LIN {X 0,Y 312.586,Z 205.55,A -85,B 0,C 180,E1 -15727.528,E2 -15727.528} C_VEL
LIN {X 0,Y 312.637,Z 205.541,A -85,B 0,C 180,E1 -15731.656,E2 -15731.656} C_VEL
LIN {X 0,Y 312.692,Z 205.534,A -85,B 0,C 180,E1 -15735.685,E2 -15735.685} C_VEL
LIN {X 0,Y 312.7,Z 205.533,A -85,B 0,C 180,E1 -15739.641,E2 -15739.641} C_VEL
LIN {X 0,Y 312.87,Z 205.509,A -85,B 0,C 180,E1 -15742.253,E2 -15742.253} C_VEL
LIN {X 0,Y 312.716,Z 205.531,A -85,B 0,C 180,E1 -15744.842,E2 -15744.842} C_VEL
LIN {X 0,Y 312.988,Z 205.497,A -85,B 0,C 180,E1 -15748.712,E2 -15748.712} C_VEL
LIN {X 0,Y 312.988,Z 205.498,A -85,B 0,C 180,E1 -15751.286,E2 -15751.286} C_VEL
LIN {X 0,Y 312.713,Z 205.533,A -85,B 0,C 180,E1 -15755.157,E2 -15755.157} C_VEL
LIN {X 0,Y 312.862,Z 205.51,A -85,B 0,C 180,E1 -15757.745,E2 -15757.745} C_VEL
LIN {X 0,Y 312.665,Z 205.535,A -85,B 0,C 180,E1 -15761.67,E2 -15761.67} C_VEL
LIN {X 0,Y 312.696,Z 205.536,A -85,B 0,C 180,E1 -15764.887,E2 -15764.887} C_VEL
LIN {X 0,Y 312.626,Z 205.542,A -85,B 0,C 180,E1 -15769.236,E2 -15769.236} C_VEL
LIN {X 0,Y 312.541,Z 205.555,A -85,B 0,C 180,E1 -15772.789,E2 -15772.789} C_VEL
LIN {X 0,Y 312.577,Z 205.551,A -85,B 0,C 180,E1 -15776.722,E2 -15776.722} C_VEL
LIN {X 0,Y 312.539,Z 205.551,A -85,B 0,C 180,E1 -15779.649,E2 -15779.649} C_VEL
LIN {X 0,Y 312.513,Z 205.554,A -85,B 0,C 180,E1 -15783.688,E2 -15783.688} C_VEL
LIN {X 0,Y 312.546,Z 205.55,A -85,B 0,C 180,E1 -15787.381,E2 -15787.381} C_VEL
LIN {X 0,Y 312.526,Z 205.555,A -85,B 0,C 180,E1 -15790.702,E2 -15790.702} C_VEL
LIN {X 0,Y 312.528,Z 205.556,A -85,B 0,C 180,E1 -15794.194,E2 -15794.194} C_VEL
LIN {X 0,Y 312.526,Z 205.554,A -85,B 0,C 180,E1 -15797.908,E2 -15797.908} C_VEL
LIN {X 0,Y 312.549,Z 205.552,A -85,B 0,C 180,E1 -15801.905,E2 -15801.905} C_VEL
LIN {X 0,Y 312.499,Z 205.558,A -85,B 0,C 180,E1 -15805.79,E2 -15805.79} C_VEL
LIN {X 0,Y 312.493,Z 205.557,A -85,B 0,C 180,E1 -15806.992,E2 -15806.992} C_VEL
LIN {X 0,Y 311.844,Z 205.642,A -85,B 0,C 180,E1 -15808.068,E2 -15808.068} C_VEL
LIN {X 0,Y 309.031,Z 205.991,A -85,B 0,C 180,E1 -15809.82,E2 -15809.82} C_VEL
LIN {X 0,Y 306.634,Z 206.291,A -85,B 0,C 180,E1 -15811.24,E2 -15811.24} C_VEL
LIN {X 0,Y 305.599,Z 206.419,A -85,B 0,C 180,E1 -15812.339,E2 -15812.339} C_VEL
LIN {X 0,Y 305.511,Z 206.427,A -85,B 0,C 180,E1 -15812.712,E2 -15812.712} C_VEL
LIN {X 0,Y 305.5,Z 206.429,A -85,B 0,C 180,E1 -15815.539,E2 -15815.539} C_VEL
LIN {X 0,Y 305.511,Z 206.43,A -85,B 0,C 180,E1 -15819.815,E2 -15819.815} C_VEL
LIN {X 0,Y 305.567,Z 206.42,A -85,B 0,C 180,E1 -15822.603,E2 -15822.603} C_VEL
LIN {X 0,Y 305.641,Z 206.411,A -85,B 0,C 180,E1 -15825.349,E2 -15825.349} C_VEL
LIN {X 0,Y 305.628,Z 206.413,A -85,B 0,C 180,E1 -15829.4,E2 -15829.4} C_VEL
LIN {X 0,Y 305.789,Z 206.394,A -85,B 0,C 180,E1 -15832.074,E2 -15832.074} C_VEL
LIN {X 0,Y 305.679,Z 206.405,A -85,B 0,C 180,E1 -15834.724,E2 -15834.724} C_VEL
LIN {X 0,Y 305.949,Z 206.372,A -85,B 0,C 180,E1 -15838.684,E2 -15838.684} C_VEL
LIN {X 0,Y 305.949,Z 206.374,A -85,B 0,C 180,E1 -15841.317,E2 -15841.317} C_VEL
LIN {X 0,Y 305.844,Z 206.385,A -85,B 0,C 180,E1 -15846.598,E2 -15846.598} C_VEL
LIN {X 0,Y 305.729,Z 206.402,A -85,B 0,C 180,E1 -15849.261,E2 -15849.261} C_VEL
LIN {X 0,Y 305.582,Z 206.421,A -85,B 0,C 180,E1 -15853.297,E2 -15853.297} C_VEL
LIN {X 0,Y 305.588,Z 206.418,A -85,B 0,C 180,E1 -15856.021,E2 -15856.021} C_VEL
LIN {X 0,Y 305.571,Z 206.423,A -85,B 0,C 180,E1 -15859.446,E2 -15859.446} C_VEL
LIN {X 0,Y 305.485,Z 206.432,A -85,B 0,C 180,E1 -15863.043,E2 -15863.043} C_VEL
LIN {X 0,Y 305.52,Z 206.425,A -85,B 0,C 180,E1 -15866.22,E2 -15866.22} C_VEL
LIN {X 0,Y 305.483,Z 206.433,A -85,B 0,C 180,E1 -15869.049,E2 -15869.049} C_VEL
LIN {X 0,Y 305.437,Z 206.436,A -85,B 0,C 180,E1 -15871.954,E2 -15871.954} C_VEL
LIN {X 0,Y 305.458,Z 206.438,A -85,B 0,C 180,E1 -15875.114,E2 -15875.114} C_VEL
LIN {X 0,Y 305.436,Z 206.437,A -85,B 0,C 180,E1 -15878.528,E2 -15878.528} C_VEL
LIN {X 0,Y 305.451,Z 206.436,A -85,B 0,C 180,E1 -15882.587,E2 -15882.587} C_VEL
LIN {X 0,Y 305.422,Z 206.438,A -85,B 0,C 180,E1 -15886.346,E2 -15886.346} C_VEL
LIN {X 0,Y 305.456,Z 206.434,A -85,B 0,C 180,E1 -15889.894,E2 -15889.894} C_VEL
LIN {X 0,Y 305.478,Z 206.434,A -85,B 0,C 180,E1 -15893.633,E2 -15893.633} C_VEL
LIN {X 0,Y 305.536,Z 206.602,A -85,B 0,C 180,E1 -15895.711,E2 -15895.711} C_VEL
LIN {X 0,Y 309.119,Z 222.623,A -85,B 0,C 180,E1 -15899.555,E2 -15899.555} C_VEL
LIN {X 0,Y 311.405,Z 233.024,A -85,B 0,C 180,E1 -15901.938,E2 -15901.938} C_VEL
LIN {X 0,Y 310.895,Z 238.703,A -85,B 0,C 180,E1 -15903.122,E2 -15903.122} C_VEL
LIN {X 0,Y 308.443,Z 258.998,A -85,B 0,C 180,E1 -15907.254,E2 -15907.254} C_VEL
LIN {X 0,Y 310.83,Z 288.757,A -85,B 0,C 180,E1 -15908.249,E2 -15908.249} C_VEL
LIN {X 0,Y 311.426,Z 296.327,A -85,B 0,C 180,E1 -15908.49,E2 -15908.49} C_VEL
LIN {X 0,Y 309.963,Z 363.951,A -85,B 0,C 180,E1 -15910.377,E2 -15910.377} C_VEL
LIN {X 0,Y 309.194,Z 377.33,A -85,B 0,C 180,E1 -15911.016,E2 -15911.016} C_VEL
LIN {X 0,Y 308.473,Z 387.934,A -85,B 0,C 180,E1 -15911.745,E2 -15911.745} C_VEL
LIN {X 0,Y 307.527,Z 400.398,A -85,B 0,C 180,E1 -15912.889,E2 -15912.889} C_VEL
LIN {X 0,Y 306.587,Z 411.617,A -85,B 0,C 180,E1 -15914.219,E2 -15914.219} C_VEL
LIN {X 0,Y 305.71,Z 421.456,A -85,B 0,C 180,E1 -15915.693,E2 -15915.693} C_VEL
LIN {X 0,Y 304.983,Z 430.461,A -85,B 0,C 180,E1 -15917.356,E2 -15917.356} C_VEL
LIN {X 0,Y 304.502,Z 437.832,A -85,B 0,C 180,E1 -15919.024,E2 -15919.024} C_VEL
LIN {X 0,Y 304.218,Z 444.937,A -85,B 0,C 180,E1 -15921.03,E2 -15921.03} C_VEL
LIN {X 0,Y 304.201,Z 451.35,A -85,B 0,C 180,E1 -15923.368,E2 -15923.368} C_VEL
LIN {X 0,Y 304.234,Z 455.384,A -85,B 0,C 180,E1 -15925.363,E2 -15925.363} C_VEL
LIN {X 0,Y 304.425,Z 458.247,A -85,B 0,C 180,E1 -15927.355,E2 -15927.355} C_VEL
LIN {X 0,Y 304.502,Z 459.525,A -85,B 0,C 180,E1 -15928.678,E2 -15928.678} C_VEL
LIN {X 0,Y 304.466,Z 460.35,A -85,B 0,C 180,E1 -15930.001,E2 -15930.001} C_VEL
LIN {X 0,Y 304.461,Z 460.719,A -85,B 0,C 180,E1 -15931.324,E2 -15931.324} C_VEL
LIN {X 0,Y 304.248,Z 460.595,A -85,B 0,C 180,E1 -15932.649,E2 -15932.649} C_VEL
LIN {X 0,Y 304.007,Z 460.044,A -85,B 0,C 180,E1 -15933.978,E2 -15933.978} C_VEL
LIN {X 0,Y 303.954,Z 458.231,A -85,B 0,C 180,E1 -15936.146,E2 -15936.146} C_VEL
LIN {X 0,Y 304.006,Z 454.659,A -85,B 0,C 180,E1 -15938.643,E2 -15938.643} C_VEL
LIN {X 0,Y 304.327,Z 450.624,A -85,B 0,C 180,E1 -15940.647,E2 -15940.647} C_VEL
LIN {X 0,Y 305.295,Z 444.466,A -85,B 0,C 180,E1 -15942.971,E2 -15942.971} C_VEL
LIN {X 0,Y 306.481,Z 437.705,A -85,B 0,C 180,E1 -15944.951,E2 -15944.951} C_VEL
LIN {X 0,Y 307.994,Z 429.456,A -85,B 0,C 180,E1 -15946.881,E2 -15946.881} C_VEL
LIN {X 0,Y 309.674,Z 420.823,A -85,B 0,C 180,E1 -15948.526,E2 -15948.526} C_VEL
LIN {X 0,Y 311.798,Z 410.405,A -85,B 0,C 180,E1 -15950.106,E2 -15950.106} C_VEL
LIN {X 0,Y 313.859,Z 398.746,A -85,B 0,C 180,E1 -15951.511,E2 -15951.511} C_VEL
LIN {X 0,Y 315.687,Z 387.145,A -85,B 0,C 180,E1 -15952.584,E2 -15952.584} C_VEL
LIN {X 0,Y 317.519,Z 374.07,A -85,B 0,C 180,E1 -15953.48,E2 -15953.48} C_VEL
LIN {X 0,Y 318.763,Z 360.739,A -85,B 0,C 180,E1 -15954.116,E2 -15954.116} C_VEL
LIN {X 0,Y 320.717,Z 321.294,A -85,B 0,C 180,E1 -15955.308,E2 -15955.308} C_VEL
LIN {X 0,Y 321.751,Z 297.702,A -85,B 0,C 180,E1 -15956.035,E2 -15956.035} C_VEL
LIN {X 0,Y 320.348,Z 281.565,A -85,B 0,C 180,E1 -15956.817,E2 -15956.817} C_VEL
LIN {X 0,Y 317.918,Z 265.294,A -85,B 0,C 180,E1 -15957.783,E2 -15957.783} C_VEL
LIN {X 0,Y 316.106,Z 255.214,A -85,B 0,C 180,E1 -15958.474,E2 -15958.474} C_VEL
LIN {X 0,Y 317.384,Z 248.061,A -85,B 0,C 180,E1 -15959.917,E2 -15959.917} C_VEL
LIN {X 0,Y 317.312,Z 245.135,A -85,B 0,C 180,E1 -15960.626,E2 -15960.626} C_VEL
LIN {X 0,Y 315.192,Z 235.048,A -85,B 0,C 180,E1 -15963.495,E2 -15963.495} C_VEL
LIN {X 0,Y 313.001,Z 227.13,A -85,B 0,C 180,E1 -15966.066,E2 -15966.066} C_VEL
LIN {X 0,Y 310.682,Z 220.037,A -85,B 0,C 180,E1 -15968.7,E2 -15968.7} C_VEL
LIN {X 0,Y 307.74,Z 212.476,A -85,B 0,C 180,E1 -15972.079,E2 -15972.079} C_VEL
LIN {X 0,Y 306.8,Z 209.817,A -85,B 0,C 180,E1 -15973.411,E2 -15973.411} C_VEL
LIN {X 0,Y 305.434,Z 206.594,A -85,B 0,C 180,E1 -15975.345,E2 -15975.345} C_VEL
LIN {X 0,Y 305.444,Z 206.434,A -85,B 0,C 180,E1 -15978.143,E2 -15978.143} C_VEL
LIN {X 0,Y 305.471,Z 206.432,A -85,B 0,C 180,E1 -15981.596,E2 -15981.596} C_VEL
LIN {X 0,Y 305.466,Z 206.433,A -85,B 0,C 180,E1 -15984.887,E2 -15984.887} C_VEL
LIN {X 0,Y 305.453,Z 206.432,A -85,B 0,C 180,E1 -15988.356,E2 -15988.356} C_VEL
LIN {X 0,Y 305.516,Z 206.425,A -85,B 0,C 180,E1 -15991.113,E2 -15991.113} C_VEL
LIN {X 0,Y 305.574,Z 206.423,A -85,B 0,C 180,E1 -15994.088,E2 -15994.088} C_VEL
LIN {X 0,Y 305.503,Z 206.43,A -85,B 0,C 180,E1 -15998.402,E2 -15998.402} C_VEL
LIN {X 0,Y 305.628,Z 206.622,A -85,B 0,C 180,E1 -16001.48,E2 -16001.48} C_VEL
LIN {X 0,Y 307.294,Z 211.058,A -85,B 0,C 180,E1 -16004.07,E2 -16004.07} C_VEL
LIN {X 0,Y 309.466,Z 216.706,A -85,B 0,C 180,E1 -16006.873,E2 -16006.873} C_VEL
LIN {X 0,Y 312.183,Z 224.834,A -85,B 0,C 180,E1 -16010.279,E2 -16010.279} C_VEL
LIN {X 0,Y 313.959,Z 231.596,A -85,B 0,C 180,E1 -16012.728,E2 -16012.728} C_VEL
LIN {X 0,Y 315.055,Z 236.534,A -85,B 0,C 180,E1 -16014.298,E2 -16014.298} C_VEL
LIN {X 0,Y 318.008,Z 242.357,A -85,B 0,C 180,E1 -16015.047,E2 -16015.047} C_VEL
LIN {X 0,Y 321.331,Z 256.287,A -85,B 0,C 180,E1 -16016.159,E2 -16016.159} C_VEL
LIN {X 0,Y 322.892,Z 264.443,A -85,B 0,C 180,E1 -16016.718,E2 -16016.718} C_VEL
LIN {X 0,Y 319.31,Z 322.49,A -85,B 0,C 180,E1 -16018.738,E2 -16018.738} C_VEL
LIN {X 0,Y 318.441,Z 335.49,A -85,B 0,C 180,E1 -16019.446,E2 -16019.446} C_VEL
LIN {X 0,Y 317.313,Z 346.446,A -85,B 0,C 180,E1 -16020.278,E2 -16020.278} C_VEL
LIN {X 0,Y 315.87,Z 357.96,A -85,B 0,C 180,E1 -16021.434,E2 -16021.434} C_VEL
LIN {X 0,Y 314.377,Z 367.881,A -85,B 0,C 180,E1 -16022.722,E2 -16022.722} C_VEL
LIN {X 0,Y 312.691,Z 376.857,A -85,B 0,C 180,E1 -16024.188,E2 -16024.188} C_VEL
LIN {X 0,Y 311.231,Z 384.199,A -85,B 0,C 180,E1 -16025.696,E2 -16025.696} C_VEL
LIN {X 0,Y 309.642,Z 391.14,A -85,B 0,C 180,E1 -16027.498,E2 -16027.498} C_VEL
LIN {X 0,Y 308.405,Z 396.181,A -85,B 0,C 180,E1 -16029.178,E2 -16029.178} C_VEL
LIN {X 0,Y 307.203,Z 400.679,A -85,B 0,C 180,E1 -16031.146,E2 -16031.146} C_VEL
LIN {X 0,Y 306.147,Z 403.971,A -85,B 0,C 180,E1 -16033.271,E2 -16033.271} C_VEL
LIN {X 0,Y 305.491,Z 405.548,A -85,B 0,C 180,E1 -16034.93,E2 -16034.93} C_VEL
LIN {X 0,Y 305.155,Z 406.152,A -85,B 0,C 180,E1 -16036.043,E2 -16036.043} C_VEL
LIN {X 0,Y 304.79,Z 406.365,A -85,B 0,C 180,E1 -16037.442,E2 -16037.442} C_VEL
LIN {X 0,Y 304.567,Z 406,A -85,B 0,C 180,E1 -16038.898,E2 -16038.898} C_VEL
LIN {X 0,Y 304.389,Z 405.081,A -85,B 0,C 180,E1 -16040.262,E2 -16040.262} C_VEL
LIN {X 0,Y 304.389,Z 402.288,A -85,B 0,C 180,E1 -16042.548,E2 -16042.548} C_VEL
LIN {X 0,Y 304.598,Z 398.51,A -85,B 0,C 180,E1 -16044.538,E2 -16044.538} C_VEL
LIN {X 0,Y 304.972,Z 392.759,A -85,B 0,C 180,E1 -16046.703,E2 -16046.703} C_VEL
LIN {X 0,Y 305.379,Z 386.42,A -85,B 0,C 180,E1 -16048.524,E2 -16048.524} C_VEL
LIN {X 0,Y 305.989,Z 378.314,A -85,B 0,C 180,E1 -16050.35,E2 -16050.35} C_VEL
LIN {X 0,Y 306.664,Z 368.955,A -85,B 0,C 180,E1 -16052.01,E2 -16052.01} C_VEL
LIN {X 0,Y 307.327,Z 359.976,A -85,B 0,C 180,E1 -16053.286,E2 -16053.286} C_VEL
LIN {X 0,Y 308.049,Z 348.466,A -85,B 0,C 180,E1 -16054.576,E2 -16054.576} C_VEL
LIN {X 0,Y 308.666,Z 335.868,A -85,B 0,C 180,E1 -16055.633,E2 -16055.633} C_VEL
LIN {X 0,Y 309.157,Z 324.141,A -85,B 0,C 180,E1 -16056.332,E2 -16056.332} C_VEL
LIN {X 0,Y 309.352,Z 311.339,A -85,B 0,C 180,E1 -16056.837,E2 -16056.837} C_VEL
LIN {X 0,Y 310.809,Z 254.755,A -85,B 0,C 180,E1 -16058.574,E2 -16058.574} C_VEL
LIN {X 0,Y 307.658,Z 232.493,A -85,B 0,C 180,E1 -16059.453,E2 -16059.453} C_VEL
LIN {X 0,Y 308.195,Z 223.036,A -85,B 0,C 180,E1 -16061.836,E2 -16061.836} C_VEL
LIN {X 0,Y 307.872,Z 218.463,A -85,B 0,C 180,E1 -16063.072,E2 -16063.072} C_VEL
LIN {X 0,Y 305.51,Z 206.606,A -85,B 0,C 180,E1 -16066.507,E2 -16066.507} C_VEL
LIN {X 0,Y 305.457,Z 206.437,A -85,B 0,C 180,E1 -16069.892,E2 -16069.892} C_VEL
LIN {X 0,Y 305.48,Z 206.436,A -85,B 0,C 180,E1 -16073.631,E2 -16073.631} C_VEL
LIN {X 0,Y 305.464,Z 206.432,A -85,B 0,C 180,E1 -16076.482,E2 -16076.482} C_VEL
LIN {X 0,Y 305.463,Z 206.438,A -85,B 0,C 180,E1 -16079.59,E2 -16079.59} C_VEL
LIN {X 0,Y 305.52,Z 206.425,A -85,B 0,C 180,E1 -16082.608,E2 -16082.608} C_VEL
LIN {X 0,Y 305.507,Z 206.432,A -85,B 0,C 180,E1 -16085.538,E2 -16085.538} C_VEL
LIN {X 0,Y 305.518,Z 206.427,A -85,B 0,C 180,E1 -16089.814,E2 -16089.814} C_VEL
LIN {X 0,Y 305.573,Z 206.419,A -85,B 0,C 180,E1 -16092.602,E2 -16092.602} C_VEL
LIN {X 0,Y 305.647,Z 206.414,A -85,B 0,C 180,E1 -16095.348,E2 -16095.348} C_VEL
LIN {X 0,Y 305.637,Z 206.414,A -85,B 0,C 180,E1 -16099.399,E2 -16099.399} C_VEL
LIN {X 0,Y 305.811,Z 206.389,A -85,B 0,C 180,E1 -16102.073,E2 -16102.073} C_VEL
LIN {X 0,Y 305.688,Z 206.406,A -85,B 0,C 180,E1 -16104.723,E2 -16104.723} C_VEL
LIN {X 0,Y 305.955,Z 206.373,A -85,B 0,C 180,E1 -16108.683,E2 -16108.683} C_VEL
LIN {X 0,Y 305.955,Z 206.374,A -85,B 0,C 180,E1 -16111.315,E2 -16111.315} C_VEL
LIN {X 0,Y 305.684,Z 206.407,A -85,B 0,C 180,E1 -16115.276,E2 -16115.276} C_VEL
LIN {X 0,Y 305.804,Z 206.389,A -85,B 0,C 180,E1 -16117.925,E2 -16117.925} C_VEL
LIN {X 0,Y 305.6,Z 206.415,A -85,B 0,C 180,E1 -16121.944,E2 -16121.944} C_VEL
LIN {X 0,Y 305.633,Z 206.414,A -85,B 0,C 180,E1 -16125.034,E2 -16125.034} C_VEL
LIN {X 0,Y 305.572,Z 206.419,A -85,B 0,C 180,E1 -16129.444,E2 -16129.444} C_VEL
LIN {X 0,Y 305.485,Z 206.432,A -85,B 0,C 180,E1 -16133.041,E2 -16133.041} C_VEL
LIN {X 0,Y 305.548,Z 206.423,A -85,B 0,C 180,E1 -16136.229,E2 -16136.229} C_VEL
LIN {X 0,Y 305.49,Z 206.431,A -85,B 0,C 180,E1 -16139.049,E2 -16139.049} C_VEL
LIN {X 0,Y 305.438,Z 206.436,A -85,B 0,C 180,E1 -16141.951,E2 -16141.951} C_VEL
LIN {X 0,Y 305.457,Z 206.434,A -85,B 0,C 180,E1 -16145.112,E2 -16145.112} C_VEL
LIN {X 0,Y 305.487,Z 206.434,A -85,B 0,C 180,E1 -16148.539,E2 -16148.539} C_VEL
LIN {X 0,Y 305.502,Z 206.431,A -85,B 0,C 180,E1 -16152.596,E2 -16152.596} C_VEL
LIN {X 0,Y 305.48,Z 206.436,A -85,B 0,C 180,E1 -16156.356,E2 -16156.356} C_VEL
LIN {X 0,Y 305.459,Z 206.434,A -85,B 0,C 180,E1 -16159.893,E2 -16159.893} C_VEL
LIN {X 0,Y 305.495,Z 206.429,A -85,B 0,C 180,E1 -16163.626,E2 -16163.626} C_VEL
LIN {X 0,Y 305.428,Z 206.437,A -85,B 0,C 180,E1 -16166.983,E2 -16166.983} C_VEL
LIN {X 0,Y 305.513,Z 206.426,A -85,B 0,C 180,E1 -16171.114,E2 -16171.114} C_VEL
LIN {X 0,Y 305.511,Z 206.427,A -85,B 0,C 180,E1 -16172.712,E2 -16172.712} C_VEL
LIN {X 0,Y 304.826,Z 206.515,A -85,B 0,C 180,E1 -16173.813,E2 -16173.813} C_VEL
LIN {X 0,Y 301.945,Z 206.872,A -85,B 0,C 180,E1 -16175.604,E2 -16175.604} C_VEL
LIN {X 0,Y 299.516,Z 207.174,A -85,B 0,C 180,E1 -16177.058,E2 -16177.058} C_VEL
LIN {X 0,Y 298.486,Z 207.305,A -85,B 0,C 180,E1 -16178.184,E2 -16178.184} C_VEL
LIN {X 0,Y 298.408,Z 207.31,A -85,B 0,C 180,E1 -16178.566,E2 -16178.566} C_VEL
LIN {X 0,Y 298.53,Z 207.299,A -85,B 0,C 180,E1 -16182.18,E2 -16182.18} C_VEL
LIN {X 0,Y 298.585,Z 207.288,A -85,B 0,C 180,E1 -16184.995,E2 -16184.995} C_VEL
LIN {X 0,Y 298.584,Z 207.29,A -85,B 0,C 180,E1 -16189.147,E2 -16189.147} C_VEL
LIN {X 0,Y 298.734,Z 207.275,A -85,B 0,C 180,E1 -16191.886,E2 -16191.886} C_VEL
LIN {X 0,Y 298.649,Z 207.281,A -85,B 0,C 180,E1 -16194.599,E2 -16194.599} C_VEL
LIN {X 0,Y 298.916,Z 207.248,A -85,B 0,C 180,E1 -16198.653,E2 -16198.653} C_VEL
LIN {X 0,Y 298.916,Z 207.25,A -85,B 0,C 180,E1 -16201.348,E2 -16201.348} C_VEL
LIN {X 0,Y 298.79,Z 207.264,A -85,B 0,C 180,E1 -16206.755,E2 -16206.755} C_VEL
LIN {X 0,Y 298.674,Z 207.283,A -85,B 0,C 180,E1 -16209.481,E2 -16209.481} C_VEL
LIN {X 0,Y 298.546,Z 207.298,A -85,B 0,C 180,E1 -16213.616,E2 -16213.616} C_VEL
LIN {X 0,Y 298.543,Z 207.294,A -85,B 0,C 180,E1 -16216.41,E2 -16216.41} C_VEL
LIN {X 0,Y 298.506,Z 207.301,A -85,B 0,C 180,E1 -16219.656,E2 -16219.656} C_VEL
LIN {X 0,Y 298.452,Z 207.308,A -85,B 0,C 180,E1 -16223.599,E2 -16223.599} C_VEL
LIN {X 0,Y 298.48,Z 207.302,A -85,B 0,C 180,E1 -16226.576,E2 -16226.576} C_VEL
LIN {X 0,Y 298.412,Z 207.313,A -85,B 0,C 180,E1 -16229.643,E2 -16229.643} C_VEL
LIN {X 0,Y 298.39,Z 207.315,A -85,B 0,C 180,E1 -16232.802,E2 -16232.802} C_VEL
LIN {X 0,Y 298.44,Z 207.31,A -85,B 0,C 180,E1 -16236.808,E2 -16236.808} C_VEL
LIN {X 0,Y 298.384,Z 207.319,A -85,B 0,C 180,E1 -16241.089,E2 -16241.089} C_VEL
LIN {X 0,Y 298.396,Z 207.317,A -85,B 0,C 180,E1 -16243.105,E2 -16243.105} C_VEL
LIN {X 0,Y 298.4,Z 207.317,A -85,B 0,C 180,E1 -16246.922,E2 -16246.922} C_VEL
LIN {X 0,Y 298.397,Z 207.317,A -85,B 0,C 180,E1 -16251.009,E2 -16251.009} C_VEL
LIN {X 0,Y 298.436,Z 207.312,A -85,B 0,C 180,E1 -16254.765,E2 -16254.765} C_VEL
LIN {X 0,Y 298.504,Z 207.599,A -85,B 0,C 180,E1 -16255.383,E2 -16255.383} C_VEL
LIN {X 0,Y 302.006,Z 223.143,A -85,B 0,C 180,E1 -16259.207,E2 -16259.207} C_VEL
LIN {X 0,Y 304.454,Z 234.529,A -85,B 0,C 180,E1 -16261.874,E2 -16261.874} C_VEL
LIN {X 0,Y 302.813,Z 247.876,A -85,B 0,C 180,E1 -16264.691,E2 -16264.691} C_VEL
LIN {X 0,Y 301.499,Z 258.879,A -85,B 0,C 180,E1 -16266.956,E2 -16266.956} C_VEL
LIN {X 0,Y 304.053,Z 291.047,A -85,B 0,C 180,E1 -16268.044,E2 -16268.044} C_VEL
LIN {X 0,Y 304.463,Z 297.206,A -85,B 0,C 180,E1 -16268.245,E2 -16268.245} C_VEL
LIN {X 0,Y 303.009,Z 362.838,A -85,B 0,C 180,E1 -16270.128,E2 -16270.128} C_VEL
LIN {X 0,Y 302.298,Z 375.668,A -85,B 0,C 180,E1 -16270.742,E2 -16270.742} C_VEL
LIN {X 0,Y 301.46,Z 387.599,A -85,B 0,C 180,E1 -16271.569,E2 -16271.569} C_VEL
LIN {X 0,Y 300.569,Z 399.224,A -85,B 0,C 180,E1 -16272.656,E2 -16272.656} C_VEL
LIN {X 0,Y 299.668,Z 409.89,A -85,B 0,C 180,E1 -16273.927,E2 -16273.927} C_VEL
LIN {X 0,Y 298.749,Z 419.496,A -85,B 0,C 180,E1 -16275.352,E2 -16275.352} C_VEL
LIN {X 0,Y 298.014,Z 428.729,A -85,B 0,C 180,E1 -16277.055,E2 -16277.055} C_VEL
LIN {X 0,Y 297.505,Z 436.289,A -85,B 0,C 180,E1 -16278.763,E2 -16278.763} C_VEL
LIN {X 0,Y 297.167,Z 443.62,A -85,B 0,C 180,E1 -16280.815,E2 -16280.815} C_VEL
LIN {X 0,Y 297.111,Z 448.509,A -85,B 0,C 180,E1 -16282.526,E2 -16282.526} C_VEL
LIN {X 0,Y 297.158,Z 453.096,A -85,B 0,C 180,E1 -16284.573,E2 -16284.573} C_VEL
LIN {X 0,Y 297.233,Z 455.45,A -85,B 0,C 180,E1 -16285.933,E2 -16285.933} C_VEL
LIN {X 0,Y 297.357,Z 457.329,A -85,B 0,C 180,E1 -16287.292,E2 -16287.292} C_VEL
LIN {X 0,Y 297.458,Z 458.678,A -85,B 0,C 180,E1 -16288.647,E2 -16288.647} C_VEL
LIN {X 0,Y 297.424,Z 459.55,A -85,B 0,C 180,E1 -16290.001,E2 -16290.001} C_VEL
LIN {X 0,Y 297.412,Z 459.991,A -85,B 0,C 180,E1 -16291.355,E2 -16291.355} C_VEL
LIN {X 0,Y 297.18,Z 459.924,A -85,B 0,C 180,E1 -16292.712,E2 -16292.712} C_VEL
LIN {X 0,Y 296.892,Z 458.511,A -85,B 0,C 180,E1 -16295.434,E2 -16295.434} C_VEL
LIN {X 0,Y 296.856,Z 457.15,A -85,B 0,C 180,E1 -16296.799,E2 -16296.799} C_VEL
LIN {X 0,Y 296.944,Z 454.273,A -85,B 0,C 180,E1 -16298.85,E2 -16298.85} C_VEL
LIN {X 0,Y 297.288,Z 450.333,A -85,B 0,C 180,E1 -16300.902,E2 -16300.902} C_VEL
LIN {X 0,Y 298.193,Z 445.244,A -85,B 0,C 180,E1 -16302.939,E2 -16302.939} C_VEL
LIN {X 0,Y 299.623,Z 437.706,A -85,B 0,C 180,E1 -16305.301,E2 -16305.301} C_VEL
LIN {X 0,Y 301.233,Z 429.528,A -85,B 0,C 180,E1 -16307.306,E2 -16307.306} C_VEL
LIN {X 0,Y 302.974,Z 421.216,A -85,B 0,C 180,E1 -16308.951,E2 -16308.951} C_VEL
LIN {X 0,Y 305.182,Z 411.1,A -85,B 0,C 180,E1 -16310.561,E2 -16310.561} C_VEL
LIN {X 0,Y 307.33,Z 399.712,A -85,B 0,C 180,E1 -16311.992,E2 -16311.992} C_VEL
LIN {X 0,Y 309.22,Z 388.71,A -85,B 0,C 180,E1 -16313.084,E2 -16313.084} C_VEL
LIN {X 0,Y 310.935,Z 377.678,A -85,B 0,C 180,E1 -16313.919,E2 -16313.919} C_VEL
LIN {X 0,Y 312.486,Z 364.01,A -85,B 0,C 180,E1 -16314.676,E2 -16314.676} C_VEL
LIN {X 0,Y 313.348,Z 350.32,A -85,B 0,C 180,E1 -16315.18,E2 -16315.18} C_VEL
LIN {X 0,Y 316.005,Z 299.425,A -85,B 0,C 180,E1 -16316.714,E2 -16316.714} C_VEL
LIN {X 0,Y 314.757,Z 283.698,A -85,B 0,C 180,E1 -16317.507,E2 -16317.507} C_VEL
LIN {X 0,Y 312.523,Z 267.935,A -85,B 0,C 180,E1 -16318.473,E2 -16318.473} C_VEL
LIN {X 0,Y 310.227,Z 254.673,A -85,B 0,C 180,E1 -16319.427,E2 -16319.427} C_VEL
LIN {X 0,Y 311.077,Z 249.985,A -85,B 0,C 180,E1 -16320.401,E2 -16320.401} C_VEL
LIN {X 0,Y 310.754,Z 246.429,A -85,B 0,C 180,E1 -16321.344,E2 -16321.344} C_VEL
LIN {X 0,Y 308.655,Z 236.658,A -85,B 0,C 180,E1 -16324.283,E2 -16324.283} C_VEL
LIN {X 0,Y 306.72,Z 229.655,A -85,B 0,C 180,E1 -16326.681,E2 -16326.681} C_VEL
LIN {X 0,Y 304.675,Z 223.49,A -85,B 0,C 180,E1 -16329.095,E2 -16329.095} C_VEL
LIN {X 0,Y 301.952,Z 216.305,A -85,B 0,C 180,E1 -16332.453,E2 -16332.453} C_VEL
LIN {X 0,Y 301.133,Z 213.981,A -85,B 0,C 180,E1 -16333.655,E2 -16333.655} C_VEL
LIN {X 0,Y 299.322,Z 210.079,A -85,B 0,C 180,E1 -16336.16,E2 -16336.16} C_VEL
LIN {X 0,Y 298.402,Z 207.38,A -85,B 0,C 180,E1 -16338.29,E2 -16338.29} C_VEL
LIN {X 0,Y 298.412,Z 207.31,A -85,B 0,C 180,E1 -16342.241,E2 -16342.241} C_VEL
LIN {X 0,Y 298.412,Z 207.313,A -85,B 0,C 180,E1 -16345.581,E2 -16345.581} C_VEL
LIN {X 0,Y 298.395,Z 207.311,A -85,B 0,C 180,E1 -16348.79,E2 -16348.79} C_VEL
LIN {X 0,Y 298.462,Z 207.309,A -85,B 0,C 180,E1 -16351.904,E2 -16351.904} C_VEL
LIN {X 0,Y 298.489,Z 207.3,A -85,B 0,C 180,E1 -16354.924,E2 -16354.924} C_VEL
LIN {X 0,Y 298.493,Z 207.498,A -85,B 0,C 180,E1 -16358.686,E2 -16358.686} C_VEL
LIN {X 0,Y 300.11,Z 211.303,A -85,B 0,C 180,E1 -16361.569,E2 -16361.569} C_VEL
LIN {X 0,Y 302.043,Z 216.312,A -85,B 0,C 180,E1 -16364.523,E2 -16364.523} C_VEL
LIN {X 0,Y 304.188,Z 222.326,A -85,B 0,C 180,E1 -16367.482,E2 -16367.482} C_VEL
LIN {X 0,Y 306.717,Z 230.133,A -85,B 0,C 180,E1 -16370.77,E2 -16370.77} C_VEL
LIN {X 0,Y 308.263,Z 236.949,A -85,B 0,C 180,E1 -16373.166,E2 -16373.166} C_VEL
LIN {X 0,Y 312.996,Z 246.172,A -85,B 0,C 180,E1 -16374.447,E2 -16374.447} C_VEL
LIN {X 0,Y 316.43,Z 261.566,A -85,B 0,C 180,E1 -16375.681,E2 -16375.681} C_VEL
LIN {X 0,Y 317.142,Z 266.341,A -85,B 0,C 180,E1 -16376.003,E2 -16376.003} C_VEL
LIN {X 0,Y 313.423,Z 323.086,A -85,B 0,C 180,E1 -16378.032,E2 -16378.032} C_VEL
LIN {X 0,Y 312.507,Z 335.54,A -85,B 0,C 180,E1 -16378.711,E2 -16378.711} C_VEL
LIN {X 0,Y 311.419,Z 346.158,A -85,B 0,C 180,E1 -16379.514,E2 -16379.514} C_VEL
LIN {X 0,Y 309.914,Z 357.516,A -85,B 0,C 180,E1 -16380.651,E2 -16380.651} C_VEL
LIN {X 0,Y 308.272,Z 367.589,A -85,B 0,C 180,E1 -16381.959,E2 -16381.959} C_VEL
LIN {X 0,Y 306.67,Z 375.822,A -85,B 0,C 180,E1 -16383.284,E2 -16383.284} C_VEL
LIN {X 0,Y 304.928,Z 384.109,A -85,B 0,C 180,E1 -16384.958,E2 -16384.958} C_VEL
LIN {X 0,Y 303.405,Z 390.75,A -85,B 0,C 180,E1 -16386.65,E2 -16386.65} C_VEL
LIN {X 0,Y 301.718,Z 396.95,A -85,B 0,C 180,E1 -16388.708,E2 -16388.708} C_VEL
LIN {X 0,Y 300.367,Z 401.538,A -85,B 0,C 180,E1 -16390.788,E2 -16390.788} C_VEL
LIN {X 0,Y 299.629,Z 403.785,A -85,B 0,C 180,E1 -16392.186,E2 -16392.186} C_VEL
LIN {X 0,Y 298.956,Z 405.444,A -85,B 0,C 180,E1 -16393.596,E2 -16393.596} C_VEL
LIN {X 0,Y 298.411,Z 406.575,A -85,B 0,C 180,E1 -16395.069,E2 -16395.069} C_VEL
LIN {X 0,Y 297.972,Z 407.048,A -85,B 0,C 180,E1 -16396.441,E2 -16396.441} C_VEL
LIN {X 0,Y 297.645,Z 406.99,A -85,B 0,C 180,E1 -16397.875,E2 -16397.875} C_VEL
LIN {X 0,Y 297.423,Z 406.355,A -85,B 0,C 180,E1 -16399.318,E2 -16399.318} C_VEL
LIN {X 0,Y 297.288,Z 405.106,A -85,B 0,C 180,E1 -16400.769,E2 -16400.769} C_VEL
LIN {X 0,Y 297.317,Z 402.372,A -85,B 0,C 180,E1 -16402.796,E2 -16402.796} C_VEL
LIN {X 0,Y 297.495,Z 399.257,A -85,B 0,C 180,E1 -16404.419,E2 -16404.419} C_VEL
LIN {X 0,Y 297.872,Z 393.545,A -85,B 0,C 180,E1 -16406.633,E2 -16406.633} C_VEL
LIN {X 0,Y 298.292,Z 387.243,A -85,B 0,C 180,E1 -16408.496,E2 -16408.496} C_VEL
LIN {X 0,Y 298.889,Z 379.151,A -85,B 0,C 180,E1 -16410.367,E2 -16410.367} C_VEL
LIN {X 0,Y 299.488,Z 371.033,A -85,B 0,C 180,E1 -16411.87,E2 -16411.87} C_VEL
LIN {X 0,Y 300.259,Z 360.929,A -85,B 0,C 180,E1 -16413.37,E2 -16413.37} C_VEL
LIN {X 0,Y 300.983,Z 349.663,A -85,B 0,C 180,E1 -16414.673,E2 -16414.673} C_VEL
LIN {X 0,Y 301.568,Z 338.856,A -85,B 0,C 180,E1 -16415.634,E2 -16415.634} C_VEL
LIN {X 0,Y 302.117,Z 326.182,A -85,B 0,C 180,E1 -16416.461,E2 -16416.461} C_VEL
LIN {X 0,Y 302.408,Z 313.068,A -85,B 0,C 180,E1 -16417.017,E2 -16417.017} C_VEL
LIN {X 0,Y 303.881,Z 255.418,A -85,B 0,C 180,E1 -16418.843,E2 -16418.843} C_VEL
LIN {X 0,Y 300.689,Z 232.571,A -85,B 0,C 180,E1 -16419.784,E2 -16419.784} C_VEL
LIN {X 0,Y 301.231,Z 221.891,A -85,B 0,C 180,E1 -16422.577,E2 -16422.577} C_VEL
LIN {X 0,Y 298.913,Z 209.734,A -85,B 0,C 180,E1 -16426.084,E2 -16426.084} C_VEL
LIN {X 0,Y 298.496,Z 207.637,A -85,B 0,C 180,E1 -16426.729,E2 -16426.729} C_VEL
LIN {X 0,Y 298.467,Z 207.336,A -85,B 0,C 180,E1 -16426.932,E2 -16426.932} C_VEL
LIN {X 0,Y 298.403,Z 207.313,A -85,B 0,C 180,E1 -16431.005,E2 -16431.005} C_VEL
LIN {X 0,Y 298.417,Z 207.313,A -85,B 0,C 180,E1 -16433.929,E2 -16433.929} C_VEL
LIN {X 0,Y 298.395,Z 207.315,A -85,B 0,C 180,E1 -16437.982,E2 -16437.982} C_VEL
LIN {X 0,Y 298.462,Z 207.307,A -85,B 0,C 180,E1 -16441.903,E2 -16441.903} C_VEL
LIN {X 0,Y 298.484,Z 207.303,A -85,B 0,C 180,E1 -16444.923,E2 -16444.923} C_VEL
LIN {X 0,Y 298.449,Z 207.311,A -85,B 0,C 180,E1 -16449.314,E2 -16449.314} C_VEL
LIN {X 0,Y 298.536,Z 207.295,A -85,B 0,C 180,E1 -16452.178,E2 -16452.178} C_VEL
LIN {X 0,Y 298.592,Z 207.29,A -85,B 0,C 180,E1 -16454.994,E2 -16454.994} C_VEL
LIN {X 0,Y 298.592,Z 207.293,A -85,B 0,C 180,E1 -16459.146,E2 -16459.146} C_VEL
LIN {X 0,Y 298.756,Z 207.268,A -85,B 0,C 180,E1 -16461.885,E2 -16461.885} C_VEL
LIN {X 0,Y 298.658,Z 207.281,A -85,B 0,C 180,E1 -16464.598,E2 -16464.598} C_VEL
LIN {X 0,Y 298.921,Z 207.249,A -85,B 0,C 180,E1 -16468.652,E2 -16468.652} C_VEL
LIN {X 0,Y 298.921,Z 207.25,A -85,B 0,C 180,E1 -16471.346,E2 -16471.346} C_VEL
LIN {X 0,Y 298.788,Z 207.267,A -85,B 0,C 180,E1 -16476.753,E2 -16476.753} C_VEL
LIN {X 0,Y 298.677,Z 207.279,A -85,B 0,C 180,E1 -16479.48,E2 -16479.48} C_VEL
LIN {X 0,Y 298.548,Z 207.294,A -85,B 0,C 180,E1 -16483.614,E2 -16483.614} C_VEL
LIN {X 0,Y 298.544,Z 207.295,A -85,B 0,C 180,E1 -16486.408,E2 -16486.408} C_VEL
LIN {X 0,Y 298.507,Z 207.299,A -85,B 0,C 180,E1 -16489.654,E2 -16489.654} C_VEL
LIN {X 0,Y 298.452,Z 207.305,A -85,B 0,C 180,E1 -16493.597,E2 -16493.597} C_VEL
LIN {X 0,Y 298.486,Z 207.305,A -85,B 0,C 180,E1 -16496.573,E2 -16496.573} C_VEL
LIN {X 0,Y 298.415,Z 207.31,A -85,B 0,C 180,E1 -16499.64,E2 -16499.64} C_VEL
LIN {X 0,Y 298.389,Z 207.316,A -85,B 0,C 180,E1 -16502.799,E2 -16502.799} C_VEL
LIN {X 0,Y 298.464,Z 207.307,A -85,B 0,C 180,E1 -16506.813,E2 -16506.813} C_VEL
LIN {X 0,Y 298.448,Z 207.306,A -85,B 0,C 180,E1 -16511.102,E2 -16511.102} C_VEL
LIN {X 0,Y 298.452,Z 207.306,A -85,B 0,C 180,E1 -16513.115,E2 -16513.115} C_VEL
LIN {X 0,Y 298.428,Z 207.309,A -85,B 0,C 180,E1 -16516.926,E2 -16516.926} C_VEL
LIN {X 0,Y 298.424,Z 207.309,A -85,B 0,C 180,E1 -16520.999,E2 -16520.999} C_VEL
LIN {X 0,Y 298.427,Z 207.311,A -85,B 0,C 180,E1 -16523.932,E2 -16523.932} C_VEL
LIN {X 0,Y 298.392,Z 207.316,A -85,B 0,C 180,E1 -16527.982,E2 -16527.982} C_VEL
LIN {X 0,Y 298.456,Z 207.308,A -85,B 0,C 180,E1 -16531.904,E2 -16531.904} C_VEL
LIN {X 0,Y 298.478,Z 207.302,A -85,B 0,C 180,E1 -16534.924,E2 -16534.924} C_VEL
LIN {X 0,Y 298.408,Z 207.31,A -85,B 0,C 180,E1 -16538.566,E2 -16538.566} C_VEL
LIN {X 0,Y 297.753,Z 207.396,A -85,B 0,C 180,E1 -16539.692,E2 -16539.692} C_VEL
LIN {X 0,Y 294.911,Z 207.749,A -85,B 0,C 180,E1 -16541.528,E2 -16541.528} C_VEL
LIN {X 0,Y 292.538,Z 208.042,A -85,B 0,C 180,E1 -16543.018,E2 -16543.018} C_VEL
LIN {X 0,Y 291.584,Z 208.163,A -85,B 0,C 180,E1 -16544.171,E2 -16544.171} C_VEL
LIN {X 0,Y 291.541,Z 208.166,A -85,B 0,C 180,E1 -16544.561,E2 -16544.561} C_VEL
LIN {X 0,Y 291.528,Z 208.168,A -85,B 0,C 180,E1 -16548.881,E2 -16548.881} C_VEL
LIN {X 0,Y 291.681,Z 208.153,A -85,B 0,C 180,E1 -16551.688,E2 -16551.688} C_VEL
LIN {X 0,Y 291.62,Z 208.157,A -85,B 0,C 180,E1 -16554.469,E2 -16554.469} C_VEL
LIN {X 0,Y 291.882,Z 208.124,A -85,B 0,C 180,E1 -16558.621,E2 -16558.621} C_VEL
LIN {X 0,Y 291.882,Z 208.126,A -85,B 0,C 180,E1 -16561.38,E2 -16561.38} C_VEL
LIN {X 0,Y 291.739,Z 208.143,A -85,B 0,C 180,E1 -16566.919,E2 -16566.919} C_VEL
LIN {X 0,Y 291.623,Z 208.159,A -85,B 0,C 180,E1 -16569.713,E2 -16569.713} C_VEL
LIN {X 0,Y 291.516,Z 208.171,A -85,B 0,C 180,E1 -16573.951,E2 -16573.951} C_VEL
LIN {X 0,Y 291.481,Z 208.175,A -85,B 0,C 180,E1 -16576.819,E2 -16576.819} C_VEL
LIN {X 0,Y 291.445,Z 208.179,A -85,B 0,C 180,E1 -16579.876,E2 -16579.876} C_VEL
LIN {X 0,Y 291.394,Z 208.185,A -85,B 0,C 180,E1 -16584.206,E2 -16584.206} C_VEL
LIN {X 0,Y 291.414,Z 208.187,A -85,B 0,C 180,E1 -16587.273,E2 -16587.273} C_VEL
LIN {X 0,Y 291.33,Z 208.193,A -85,B 0,C 180,E1 -16590.438,E2 -16590.438} C_VEL
LIN {X 0,Y 291.34,Z 208.193,A -85,B 0,C 180,E1 -16593.7,E2 -16593.7} C_VEL
LIN {X 0,Y 291.368,Z 208.192,A -85,B 0,C 180,E1 -16597.254,E2 -16597.254} C_VEL
LIN {X 0,Y 291.329,Z 208.195,A -85,B 0,C 180,E1 -16600.644,E2 -16600.644} C_VEL
LIN {X 0,Y 291.287,Z 208.199,A -85,B 0,C 180,E1 -16604.403,E2 -16604.403} C_VEL
LIN {X 0,Y 291.324,Z 208.195,A -85,B 0,C 180,E1 -16608.406,E2 -16608.406} C_VEL
LIN {X 0,Y 291.346,Z 208.195,A -85,B 0,C 180,E1 -16611.159,E2 -16611.159} C_VEL
LIN {X 0,Y 291.417,Z 208.319,A -85,B 0,C 180,E1 -16614.957,E2 -16614.957} C_VEL
LIN {X 0,Y 294.6,Z 222.569,A -85,B 0,C 180,E1 -16618.583,E2 -16618.583} C_VEL
LIN {X 0,Y 297.158,Z 234.002,A -85,B 0,C 180,E1 -16621.345,E2 -16621.345} C_VEL
LIN {X 0,Y 297.474,Z 235.968,A -85,B 0,C 180,E1 -16621.804,E2 -16621.804} C_VEL
LIN {X 0,Y 294.864,Z 255.874,A -85,B 0,C 180,E1 -16626.098,E2 -16626.098} C_VEL
LIN {X 0,Y 294.548,Z 258.705,A -85,B 0,C 180,E1 -16626.635,E2 -16626.635} C_VEL
LIN {X 0,Y 297.025,Z 290.847,A -85,B 0,C 180,E1 -16627.756,E2 -16627.756} C_VEL
LIN {X 0,Y 297.514,Z 297.833,A -85,B 0,C 180,E1 -16627.99,E2 -16627.99} C_VEL
LIN {X 0,Y 296.009,Z 362.76,A -85,B 0,C 180,E1 -16629.909,E2 -16629.909} C_VEL
LIN {X 0,Y 295.297,Z 375.434,A -85,B 0,C 180,E1 -16630.538,E2 -16630.538} C_VEL
LIN {X 0,Y 294.436,Z 387.253,A -85,B 0,C 180,E1 -16631.383,E2 -16631.383} C_VEL
LIN {X 0,Y 293.47,Z 399.621,A -85,B 0,C 180,E1 -16632.583,E2 -16632.583} C_VEL
LIN {X 0,Y 292.502,Z 410.674,A -85,B 0,C 180,E1 -16633.966,E2 -16633.966} C_VEL
LIN {X 0,Y 291.492,Z 421.519,A -85,B 0,C 180,E1 -16635.693,E2 -16635.693} C_VEL
LIN {X 0,Y 290.777,Z 430.291,A -85,B 0,C 180,E1 -16637.437,E2 -16637.437} C_VEL
LIN {X 0,Y 290.259,Z 438.71,A -85,B 0,C 180,E1 -16639.538,E2 -16639.538} C_VEL
LIN {X 0,Y 290.052,Z 445.401,A -85,B 0,C 180,E1 -16641.642,E2 -16641.642} C_VEL
LIN {X 0,Y 290.153,Z 450.627,A -85,B 0,C 180,E1 -16643.763,E2 -16643.763} C_VEL
LIN {X 0,Y 290.177,Z 454.448,A -85,B 0,C 180,E1 -16645.834,E2 -16645.834} C_VEL
LIN {X 0,Y 290.292,Z 456.375,A -85,B 0,C 180,E1 -16647.226,E2 -16647.226} C_VEL
LIN {X 0,Y 290.414,Z 457.821,A -85,B 0,C 180,E1 -16648.614,E2 -16648.614} C_VEL
LIN {X 0,Y 290.383,Z 458.739,A -85,B 0,C 180,E1 -16650.001,E2 -16650.001} C_VEL
LIN {X 0,Y 290.363,Z 459.225,A -85,B 0,C 180,E1 -16651.388,E2 -16651.388} C_VEL
LIN {X 0,Y 290.093,Z 459.247,A -85,B 0,C 180,E1 -16652.778,E2 -16652.778} C_VEL
LIN {X 0,Y 289.851,Z 458.793,A -85,B 0,C 180,E1 -16654.172,E2 -16654.172} C_VEL
LIN {X 0,Y 289.78,Z 457.526,A -85,B 0,C 180,E1 -16656.078,E2 -16656.078} C_VEL
LIN {X 0,Y 289.835,Z 454.899,A -85,B 0,C 180,E1 -16658.367,E2 -16658.367} C_VEL
LIN {X 0,Y 290.087,Z 451.42,A -85,B 0,C 180,E1 -16660.47,E2 -16660.47} C_VEL
LIN {X 0,Y 290.869,Z 446.874,A -85,B 0,C 180,E1 -16662.561,E2 -16662.561} C_VEL
LIN {X 0,Y 291.992,Z 441.115,A -85,B 0,C 180,E1 -16664.64,E2 -16664.64} C_VEL
LIN {X 0,Y 293.624,Z 433.645,A -85,B 0,C 180,E1 -16666.779,E2 -16666.779} C_VEL
LIN {X 0,Y 295.505,Z 425.041,A -85,B 0,C 180,E1 -16668.728,E2 -16668.728} C_VEL
LIN {X 0,Y 297.852,Z 414.973,A -85,B 0,C 180,E1 -16670.548,E2 -16670.548} C_VEL
LIN {X 0,Y 300.263,Z 403.528,A -85,B 0,C 180,E1 -16672.175,E2 -16672.175} C_VEL
LIN {X 0,Y 302.485,Z 392.047,A -85,B 0,C 180,E1 -16673.447,E2 -16673.447} C_VEL
LIN {X 0,Y 304.546,Z 379.952,A -85,B 0,C 180,E1 -16674.454,E2 -16674.454} C_VEL
LIN {X 0,Y 306.257,Z 366.887,A -85,B 0,C 180,E1 -16675.258,E2 -16675.258} C_VEL
LIN {X 0,Y 307.375,Z 352.431,A -85,B 0,C 180,E1 -16675.855,E2 -16675.855} C_VEL
LIN {X 0,Y 310.308,Z 300.001,A -85,B 0,C 180,E1 -16677.497,E2 -16677.497} C_VEL
LIN {X 0,Y 309.13,Z 284.637,A -85,B 0,C 180,E1 -16678.303,E2 -16678.303} C_VEL
LIN {X 0,Y 306.815,Z 267.709,A -85,B 0,C 180,E1 -16679.39,E2 -16679.39} C_VEL
LIN {X 0,Y 304.423,Z 254.107,A -85,B 0,C 180,E1 -16680.462,E2 -16680.462} C_VEL
LIN {X 0,Y 304.766,Z 251.952,A -85,B 0,C 180,E1 -16680.92,E2 -16680.92} C_VEL
LIN {X 0,Y 303.631,Z 245.049,A -85,B 0,C 180,E1 -16682.939,E2 -16682.939} C_VEL
LIN {X 0,Y 301.771,Z 236.896,A -85,B 0,C 180,E1 -16685.608,E2 -16685.608} C_VEL
LIN {X 0,Y 299.442,Z 228.979,A -85,B 0,C 180,E1 -16688.63,E2 -16688.63} C_VEL
LIN {X 0,Y 296.659,Z 221.365,A -85,B 0,C 180,E1 -16692.193,E2 -16692.193} C_VEL
LIN {X 0,Y 295.109,Z 217.463,A -85,B 0,C 180,E1 -16694.401,E2 -16694.401} C_VEL
LIN {X 0,Y 293.065,Z 212.243,A -85,B 0,C 180,E1 -16698.024,E2 -16698.024} C_VEL
LIN {X 0,Y 291.39,Z 208.307,A -85,B 0,C 180,E1 -16702.337,E2 -16702.337} C_VEL
LIN {X 0,Y 291.348,Z 208.189,A -85,B 0,C 180,E1 -16706.301,E2 -16706.301} C_VEL
LIN {X 0,Y 291.387,Z 208.186,A -85,B 0,C 180,E1 -16710.261,E2 -16710.261} C_VEL
LIN {X 0,Y 291.431,Z 208.266,A -85,B 0,C 180,E1 -16714.273,E2 -16714.273} C_VEL
LIN {X 0,Y 292.272,Z 210.852,A -85,B 0,C 180,E1 -16717.372,E2 -16717.372} C_VEL
LIN {X 0,Y 293.913,Z 214.362,A -85,B 0,C 180,E1 -16720.441,E2 -16720.441} C_VEL
LIN {X 0,Y 295.757,Z 218.854,A -85,B 0,C 180,E1 -16723.431,E2 -16723.431} C_VEL
LIN {X 0,Y 297.695,Z 224.226,A -85,B 0,C 180,E1 -16726.344,E2 -16726.344} C_VEL
LIN {X 0,Y 299.639,Z 230.435,A -85,B 0,C 180,E1 -16729.184,E2 -16729.184} C_VEL
LIN {X 0,Y 301.065,Z 235.478,A -85,B 0,C 180,E1 -16731.242,E2 -16731.242} C_VEL
LIN {X 0,Y 301.683,Z 237.727,A -85,B 0,C 180,E1 -16732.002,E2 -16732.002} C_VEL
LIN {X 0,Y 308.082,Z 250.149,A -85,B 0,C 180,E1 -16733.824,E2 -16733.824} C_VEL
LIN {X 0,Y 311.466,Z 266.319,A -85,B 0,C 180,E1 -16735.152,E2 -16735.152} C_VEL
LIN {X 0,Y 311.261,Z 271.582,A -85,B 0,C 180,E1 -16735.369,E2 -16735.369} C_VEL
LIN {X 0,Y 307.619,Z 323.983,A -85,B 0,C 180,E1 -16737.299,E2 -16737.299} C_VEL
LIN {X 0,Y 306.573,Z 336.831,A -85,B 0,C 180,E1 -16738.029,E2 -16738.029} C_VEL
LIN {X 0,Y 305.18,Z 349.012,A -85,B 0,C 180,E1 -16739.01,E2 -16739.01} C_VEL
LIN {X 0,Y 303.581,Z 359.983,A -85,B 0,C 180,E1 -16740.179,E2 -16740.179} C_VEL
LIN {X 0,Y 301.869,Z 369.68,A -85,B 0,C 180,E1 -16741.5,E2 -16741.5} C_VEL
LIN {X 0,Y 299.991,Z 378.522,A -85,B 0,C 180,E1 -16743.021,E2 -16743.021} C_VEL
LIN {X 0,Y 298.191,Z 386.387,A -85,B 0,C 180,E1 -16744.731,E2 -16744.731} C_VEL
LIN {X 0,Y 296.198,Z 393.802,A -85,B 0,C 180,E1 -16746.813,E2 -16746.813} C_VEL
LIN {X 0,Y 294.546,Z 399.414,A -85,B 0,C 180,E1 -16748.922,E2 -16748.922} C_VEL
LIN {X 0,Y 293.191,Z 403.515,A -85,B 0,C 180,E1 -16751.055,E2 -16751.055} C_VEL
LIN {X 0,Y 292.423,Z 405.442,A -85,B 0,C 180,E1 -16752.491,E2 -16752.491} C_VEL
LIN {X 0,Y 291.761,Z 406.807,A -85,B 0,C 180,E1 -16753.938,E2 -16753.938} C_VEL
LIN {X 0,Y 291.25,Z 407.597,A -85,B 0,C 180,E1 -16755.392,E2 -16755.392} C_VEL
LIN {X 0,Y 290.807,Z 407.808,A -85,B 0,C 180,E1 -16756.858,E2 -16756.858} C_VEL
LIN {X 0,Y 290.367,Z 406.944,A -85,B 0,C 180,E1 -16759.273,E2 -16759.273} C_VEL
LIN {X 0,Y 290.19,Z 403.983,A -85,B 0,C 180,E1 -16762.048,E2 -16762.048} C_VEL
LIN {X 0,Y 290.386,Z 399.968,A -85,B 0,C 180,E1 -16764.294,E2 -16764.294} C_VEL
LIN {X 0,Y 290.775,Z 394.198,A -85,B 0,C 180,E1 -16766.582,E2 -16766.582} C_VEL
LIN {X 0,Y 291.189,Z 387.981,A -85,B 0,C 180,E1 -16768.468,E2 -16768.468} C_VEL
LIN {X 0,Y 291.802,Z 379.93,A -85,B 0,C 180,E1 -16770.382,E2 -16770.382} C_VEL
LIN {X 0,Y 292.416,Z 371.876,A -85,B 0,C 180,E1 -16771.92,E2 -16771.92} C_VEL
LIN {X 0,Y 293.187,Z 361.84,A -85,B 0,C 180,E1 -16773.458,E2 -16773.458} C_VEL
LIN {X 0,Y 293.932,Z 350.528,A -85,B 0,C 180,E1 -16774.809,E2 -16774.809} C_VEL
LIN {X 0,Y 294.596,Z 338.643,A -85,B 0,C 180,E1 -16775.886,E2 -16775.886} C_VEL
LIN {X 0,Y 295.131,Z 326.337,A -85,B 0,C 180,E1 -16776.694,E2 -16776.694} C_VEL
LIN {X 0,Y 295.414,Z 312.985,A -85,B 0,C 180,E1 -16777.267,E2 -16777.267} C_VEL
LIN {X 0,Y 296.933,Z 256.216,A -85,B 0,C 180,E1 -16779.114,E2 -16779.114} C_VEL
LIN {X 0,Y 293.74,Z 232.925,A -85,B 0,C 180,E1 -16780.094,E2 -16780.094} C_VEL
LIN {X 0,Y 294.274,Z 224.761,A -85,B 0,C 180,E1 -16782.237,E2 -16782.237} C_VEL
LIN {X 0,Y 293.683,Z 219.879,A -85,B 0,C 180,E1 -16783.623,E2 -16783.623} C_VEL
LIN {X 0,Y 291.474,Z 208.507,A -85,B 0,C 180,E1 -16787.015,E2 -16787.015} C_VEL
LIN {X 0,Y 291.361,Z 208.192,A -85,B 0,C 180,E1 -16787.514,E2 -16787.514} C_VEL
LIN {X 0,Y 291.352,Z 208.192,A -85,B 0,C 180,E1 -16791.157,E2 -16791.157} C_VEL
LIN {X 0,Y 291.36,Z 208.189,A -85,B 0,C 180,E1 -16794.625,E2 -16794.625} C_VEL
LIN {X 0,Y 291.372,Z 208.19,A -85,B 0,C 180,E1 -16797.95,E2 -16797.95} C_VEL
LIN {X 0,Y 291.381,Z 208.189,A -85,B 0,C 180,E1 -16801.157,E2 -16801.157} C_VEL
LIN {X 0,Y 291.415,Z 208.182,A -85,B 0,C 180,E1 -16804.271,E2 -16804.271} C_VEL
LIN {X 0,Y 291.38,Z 208.191,A -85,B 0,C 180,E1 -16807.299,E2 -16807.299} C_VEL
LIN {X 0,Y 291.457,Z 208.177,A -85,B 0,C 180,E1 -16810.269,E2 -16810.269} C_VEL
LIN {X 0,Y 291.553,Z 208.165,A -85,B 0,C 180,E1 -16814.623,E2 -16814.623} C_VEL
LIN {X 0,Y 291.535,Z 208.169,A -85,B 0,C 180,E1 -16818.88,E2 -16818.88} C_VEL
LIN {X 0,Y 291.707,Z 208.147,A -85,B 0,C 180,E1 -16821.688,E2 -16821.688} C_VEL
LIN {X 0,Y 291.629,Z 208.156,A -85,B 0,C 180,E1 -16824.467,E2 -16824.467} C_VEL
LIN {X 0,Y 291.887,Z 208.124,A -85,B 0,C 180,E1 -16828.619,E2 -16828.619} C_VEL
LIN {X 0,Y 291.887,Z 208.126,A -85,B 0,C 180,E1 -16831.379,E2 -16831.379} C_VEL
LIN {X 0,Y 291.738,Z 208.147,A -85,B 0,C 180,E1 -16836.917,E2 -16836.917} C_VEL
LIN {X 0,Y 291.625,Z 208.156,A -85,B 0,C 180,E1 -16839.711,E2 -16839.711} C_VEL
LIN {X 0,Y 291.518,Z 208.169,A -85,B 0,C 180,E1 -16843.949,E2 -16843.949} C_VEL
LIN {X 0,Y 291.483,Z 208.178,A -85,B 0,C 180,E1 -16846.817,E2 -16846.817} C_VEL
LIN {X 0,Y 291.446,Z 208.178,A -85,B 0,C 180,E1 -16849.874,E2 -16849.874} C_VEL
LIN {X 0,Y 291.395,Z 208.186,A -85,B 0,C 180,E1 -16854.204,E2 -16854.204} C_VEL
LIN {X 0,Y 291.42,Z 208.182,A -85,B 0,C 180,E1 -16857.27,E2 -16857.27} C_VEL
LIN {X 0,Y 291.332,Z 208.196,A -85,B 0,C 180,E1 -16860.436,E2 -16860.436} C_VEL
LIN {X 0,Y 291.339,Z 208.191,A -85,B 0,C 180,E1 -16863.698,E2 -16863.698} C_VEL
LIN {X 0,Y 291.398,Z 208.185,A -85,B 0,C 180,E1 -16867.261,E2 -16867.261} C_VEL
LIN {X 0,Y 291.398,Z 208.187,A -85,B 0,C 180,E1 -16870.63,E2 -16870.63} C_VEL
LIN {X 0,Y 291.346,Z 208.196,A -85,B 0,C 180,E1 -16874.389,E2 -16874.389} C_VEL
LIN {X 0,Y 291.35,Z 208.194,A -85,B 0,C 180,E1 -16878.397,E2 -16878.397} C_VEL
LIN {X 0,Y 291.373,Z 208.187,A -85,B 0,C 180,E1 -16881.162,E2 -16881.162} C_VEL
LIN {X 0,Y 291.379,Z 208.189,A -85,B 0,C 180,E1 -16884.629,E2 -16884.629} C_VEL
LIN {X 0,Y 291.368,Z 208.191,A -85,B 0,C 180,E1 -16887.951,E2 -16887.951} C_VEL
LIN {X 0,Y 291.375,Z 208.187,A -85,B 0,C 180,E1 -16891.158,E2 -16891.158} C_VEL
LIN {X 0,Y 291.409,Z 208.186,A -85,B 0,C 180,E1 -16894.272,E2 -16894.272} C_VEL
LIN {X 0,Y 291.374,Z 208.187,A -85,B 0,C 180,E1 -16897.3,E2 -16897.3} C_VEL
LIN {X 0,Y 291.45,Z 208.181,A -85,B 0,C 180,E1 -16900.27,E2 -16900.27} C_VEL
LIN {X 0,Y 291.541,Z 208.166,A -85,B 0,C 180,E1 -16904.561,E2 -16904.561} C_VEL
LIN {X 0,Y 291.283,Z 208.202,A -85,B 0,C 180,E1 -16905.333,E2 -16905.333} C_VEL
LIN {X 0,Y 289.952,Z 208.371,A -85,B 0,C 180,E1 -16906.471,E2 -16906.471} C_VEL
LIN {X 0,Y 285.595,Z 208.911,A -85,B 0,C 180,E1 -16909.116,E2 -16909.116} C_VEL
LIN {X 0,Y 284.616,Z 209.031,A -85,B 0,C 180,E1 -16910.299,E2 -16910.299} C_VEL
LIN {X 0,Y 284.579,Z 209.034,A -85,B 0,C 180,E1 -16910.7,E2 -16910.7} C_VEL
LIN {X 0,Y 284.679,Z 209.021,A -85,B 0,C 180,E1 -16912.91,E2 -16912.91} C_VEL
LIN {X 0,Y 284.848,Z 209,A -85,B 0,C 180,E1 -16918.587,E2 -16918.587} C_VEL
LIN {X 0,Y 284.848,Z 209.003,A -85,B 0,C 180,E1 -16921.414,E2 -16921.414} C_VEL
LIN {X 0,Y 284.691,Z 209.021,A -85,B 0,C 180,E1 -16927.091,E2 -16927.091} C_VEL
LIN {X 0,Y 284.56,Z 209.037,A -85,B 0,C 180,E1 -16929.956,E2 -16929.956} C_VEL
LIN {X 0,Y 284.475,Z 209.047,A -85,B 0,C 180,E1 -16934.304,E2 -16934.304} C_VEL
LIN {X 0,Y 284.419,Z 209.057,A -85,B 0,C 180,E1 -16937.249,E2 -16937.249} C_VEL
LIN {X 0,Y 284.373,Z 209.059,A -85,B 0,C 180,E1 -16940.243,E2 -16940.243} C_VEL
LIN {X 0,Y 284.364,Z 209.062,A -85,B 0,C 180,E1 -16943.876,E2 -16943.876} C_VEL
LIN {X 0,Y 284.389,Z 209.061,A -85,B 0,C 180,E1 -16947.174,E2 -16947.174} C_VEL
LIN {X 0,Y 284.289,Z 209.074,A -85,B 0,C 180,E1 -16951.276,E2 -16951.276} C_VEL
LIN {X 0,Y 284.337,Z 209.067,A -85,B 0,C 180,E1 -16955.349,E2 -16955.349} C_VEL
LIN {X 0,Y 284.304,Z 209.068,A -85,B 0,C 180,E1 -16958.171,E2 -16958.171} C_VEL
LIN {X 0,Y 284.266,Z 209.073,A -85,B 0,C 180,E1 -16962.126,E2 -16962.126} C_VEL
LIN {X 0,Y 284.252,Z 209.075,A -85,B 0,C 180,E1 -16966.191,E2 -16966.191} C_VEL
LIN {X 0,Y 284.304,Z 209.069,A -85,B 0,C 180,E1 -16970.025,E2 -16970.025} C_VEL
LIN {X 0,Y 284.388,Z 209.169,A -85,B 0,C 180,E1 -16974.558,E2 -16974.558} C_VEL
LIN {X 0,Y 287.416,Z 222.883,A -85,B 0,C 180,E1 -16978.16,E2 -16978.16} C_VEL
LIN {X 0,Y 290.356,Z 236.157,A -85,B 0,C 180,E1 -16981.444,E2 -16981.444} C_VEL
LIN {X 0,Y 290.152,Z 239.545,A -85,B 0,C 180,E1 -16982.209,E2 -16982.209} C_VEL
LIN {X 0,Y 287.627,Z 258.042,A -85,B 0,C 180,E1 -16986.273,E2 -16986.273} C_VEL
LIN {X 0,Y 289.787,Z 288.75,A -85,B 0,C 180,E1 -16987.385,E2 -16987.385} C_VEL
LIN {X 0,Y 290.584,Z 297.879,A -85,B 0,C 180,E1 -16987.706,E2 -16987.706} C_VEL
LIN {X 0,Y 289.021,Z 362.514,A -85,B 0,C 180,E1 -16989.681,E2 -16989.681} C_VEL
LIN {X 0,Y 288.292,Z 375.037,A -85,B 0,C 180,E1 -16990.324,E2 -16990.324} C_VEL
LIN {X 0,Y 287.543,Z 385.781,A -85,B 0,C 180,E1 -16991.105,E2 -16991.105} C_VEL
LIN {X 0,Y 286.642,Z 396.744,A -85,B 0,C 180,E1 -16992.154,E2 -16992.154} C_VEL
LIN {X 0,Y 285.662,Z 407.951,A -85,B 0,C 180,E1 -16993.53,E2 -16993.53} C_VEL
LIN {X 0,Y 284.632,Z 418.469,A -85,B 0,C 180,E1 -16995.158,E2 -16995.158} C_VEL
LIN {X 0,Y 283.977,Z 426.843,A -85,B 0,C 180,E1 -16996.767,E2 -16996.767} C_VEL
LIN {X 0,Y 283.334,Z 435.885,A -85,B 0,C 180,E1 -16998.918,E2 -16998.918} C_VEL
LIN {X 0,Y 283.036,Z 442.989,A -85,B 0,C 180,E1 -17001.073,E2 -17001.073} C_VEL
LIN {X 0,Y 283.03,Z 448.838,A -85,B 0,C 180,E1 -17003.345,E2 -17003.345} C_VEL
LIN {X 0,Y 283.123,Z 453.393,A -85,B 0,C 180,E1 -17005.73,E2 -17005.73} C_VEL
LIN {X 0,Y 283.23,Z 455.38,A -85,B 0,C 180,E1 -17007.156,E2 -17007.156} C_VEL
LIN {X 0,Y 283.37,Z 456.905,A -85,B 0,C 180,E1 -17008.58,E2 -17008.58} C_VEL
LIN {X 0,Y 283.343,Z 457.915,A -85,B 0,C 180,E1 -17010.001,E2 -17010.001} C_VEL
LIN {X 0,Y 283.312,Z 458.453,A -85,B 0,C 180,E1 -17011.422,E2 -17011.422} C_VEL
LIN {X 0,Y 283.03,Z 458.533,A -85,B 0,C 180,E1 -17012.848,E2 -17012.848} C_VEL
LIN {X 0,Y 282.775,Z 458.17,A -85,B 0,C 180,E1 -17014.277,E2 -17014.277} C_VEL
LIN {X 0,Y 282.695,Z 457.108,A -85,B 0,C 180,E1 -17016.046,E2 -17016.046} C_VEL
LIN {X 0,Y 282.757,Z 454.481,A -85,B 0,C 180,E1 -17018.578,E2 -17018.578} C_VEL
LIN {X 0,Y 283.061,Z 451.136,A -85,B 0,C 180,E1 -17020.733,E2 -17020.733} C_VEL
LIN {X 0,Y 283.92,Z 446.708,A -85,B 0,C 180,E1 -17022.873,E2 -17022.873} C_VEL
LIN {X 0,Y 285.33,Z 439.999,A -85,B 0,C 180,E1 -17025.355,E2 -17025.355} C_VEL
LIN {X 0,Y 287.086,Z 432.781,A -85,B 0,C 180,E1 -17027.452,E2 -17027.452} C_VEL
LIN {X 0,Y 289.192,Z 423.816,A -85,B 0,C 180,E1 -17029.522,E2 -17029.522} C_VEL
LIN {X 0,Y 291.767,Z 413.648,A -85,B 0,C 180,E1 -17031.367,E2 -17031.367} C_VEL
LIN {X 0,Y 294.052,Z 403.313,A -85,B 0,C 180,E1 -17032.855,E2 -17032.855} C_VEL
LIN {X 0,Y 296.372,Z 391.946,A -85,B 0,C 180,E1 -17034.146,E2 -17034.146} C_VEL
LIN {X 0,Y 298.697,Z 379.071,A -85,B 0,C 180,E1 -17035.244,E2 -17035.244} C_VEL
LIN {X 0,Y 300.483,Z 366.118,A -85,B 0,C 180,E1 -17036.058,E2 -17036.058} C_VEL
LIN {X 0,Y 301.685,Z 351.865,A -85,B 0,C 180,E1 -17036.663,E2 -17036.663} C_VEL
LIN {X 0,Y 304.73,Z 300.743,A -85,B 0,C 180,E1 -17038.3,E2 -17038.3} C_VEL
LIN {X 0,Y 303.552,Z 285.108,A -85,B 0,C 180,E1 -17039.168,E2 -17039.168} C_VEL
LIN {X 0,Y 301.201,Z 267.676,A -85,B 0,C 180,E1 -17040.358,E2 -17040.358} C_VEL
LIN {X 0,Y 298.834,Z 254.972,A -85,B 0,C 180,E1 -17041.406,E2 -17041.406} C_VEL
LIN {X 0,Y 298.393,Z 253.219,A -85,B 0,C 180,E1 -17041.689,E2 -17041.689} C_VEL
LIN {X 0,Y 296.607,Z 243.84,A -85,B 0,C 180,E1 -17044.658,E2 -17044.658} C_VEL
LIN {X 0,Y 294.547,Z 235.984,A -85,B 0,C 180,E1 -17047.559,E2 -17047.559} C_VEL
LIN {X 0,Y 292.826,Z 230.722,A -85,B 0,C 180,E1 -17049.823,E2 -17049.823} C_VEL
LIN {X 0,Y 290.374,Z 223.647,A -85,B 0,C 180,E1 -17053.439,E2 -17053.439} C_VEL
LIN {X 0,Y 288.209,Z 218.466,A -85,B 0,C 180,E1 -17056.938,E2 -17056.938} C_VEL
LIN {X 0,Y 287.014,Z 215.676,A -85,B 0,C 180,E1 -17059.384,E2 -17059.384} C_VEL
LIN {X 0,Y 286.131,Z 213.248,A -85,B 0,C 180,E1 -17062.116,E2 -17062.116} C_VEL
LIN {X 0,Y 285.202,Z 211.691,A -85,B 0,C 180,E1 -17065.474,E2 -17065.474} C_VEL
LIN {X 0,Y 285.016,Z 211.355,A -85,B 0,C 180,E1 -17069.66,E2 -17069.66} C_VEL
LIN {X 0,Y 285.89,Z 212.634,A -85,B 0,C 180,E1 -17073.736,E2 -17073.736} C_VEL
LIN {X 0,Y 286.775,Z 215.132,A -85,B 0,C 180,E1 -17076.913,E2 -17076.913} C_VEL
LIN {X 0,Y 288.262,Z 218.456,A -85,B 0,C 180,E1 -17080.042,E2 -17080.042} C_VEL
LIN {X 0,Y 290,Z 222.797,A -85,B 0,C 180,E1 -17083.093,E2 -17083.093} C_VEL
LIN {X 0,Y 291.854,Z 228.055,A -85,B 0,C 180,E1 -17086.065,E2 -17086.065} C_VEL
LIN {X 0,Y 293.716,Z 234.15,A -85,B 0,C 180,E1 -17088.964,E2 -17088.964} C_VEL
LIN {X 0,Y 294.931,Z 238.179,A -85,B 0,C 180,E1 -17090.629,E2 -17090.629} C_VEL
LIN {X 0,Y 299.516,Z 246.528,A -85,B 0,C 180,E1 -17092.076,E2 -17092.076} C_VEL
LIN {X 0,Y 303.245,Z 254.182,A -85,B 0,C 180,E1 -17093.178,E2 -17093.178} C_VEL
LIN {X 0,Y 306.052,Z 268.866,A -85,B 0,C 180,E1 -17094.411,E2 -17094.411} C_VEL
LIN {X 0,Y 301.914,Z 325.201,A -85,B 0,C 180,E1 -17096.538,E2 -17096.538} C_VEL
LIN {X 0,Y 300.862,Z 337.25,A -85,B 0,C 180,E1 -17097.238,E2 -17097.238} C_VEL
LIN {X 0,Y 299.49,Z 348.582,A -85,B 0,C 180,E1 -17098.15,E2 -17098.15} C_VEL
LIN {X 0,Y 297.802,Z 359.622,A -85,B 0,C 180,E1 -17099.323,E2 -17099.323} C_VEL
LIN {X 0,Y 295.791,Z 370.197,A -85,B 0,C 180,E1 -17100.783,E2 -17100.783} C_VEL
LIN {X 0,Y 293.724,Z 379.44,A -85,B 0,C 180,E1 -17102.399,E2 -17102.399} C_VEL
LIN {X 0,Y 291.788,Z 387.291,A -85,B 0,C 180,E1 -17104.143,E2 -17104.143} C_VEL
LIN {X 0,Y 289.815,Z 394.273,A -85,B 0,C 180,E1 -17106.144,E2 -17106.144} C_VEL
LIN {X 0,Y 288.445,Z 398.541,A -85,B 0,C 180,E1 -17107.701,E2 -17107.701} C_VEL
LIN {X 0,Y 286.84,Z 403.081,A -85,B 0,C 180,E1 -17109.875,E2 -17109.875} C_VEL
LIN {X 0,Y 286.007,Z 405.314,A -85,B 0,C 180,E1 -17111.336,E2 -17111.336} C_VEL
LIN {X 0,Y 285.208,Z 406.951,A -85,B 0,C 180,E1 -17112.813,E2 -17112.813} C_VEL
LIN {X 0,Y 284.578,Z 408.03,A -85,B 0,C 180,E1 -17114.297,E2 -17114.297} C_VEL
LIN {X 0,Y 284.048,Z 408.508,A -85,B 0,C 180,E1 -17115.792,E2 -17115.792} C_VEL
LIN {X 0,Y 283.634,Z 408.437,A -85,B 0,C 180,E1 -17117.297,E2 -17117.297} C_VEL
LIN {X 0,Y 283.26,Z 407.314,A -85,B 0,C 180,E1 -17119.468,E2 -17119.468} C_VEL
LIN {X 0,Y 283.099,Z 404.701,A -85,B 0,C 180,E1 -17121.862,E2 -17121.862} C_VEL
LIN {X 0,Y 283.304,Z 400.682,A -85,B 0,C 180,E1 -17124.161,E2 -17124.161} C_VEL
LIN {X 0,Y 283.662,Z 394.971,A -85,B 0,C 180,E1 -17126.484,E2 -17126.484} C_VEL
LIN {X 0,Y 284.084,Z 388.692,A -85,B 0,C 180,E1 -17128.439,E2 -17128.439} C_VEL
LIN {X 0,Y 284.591,Z 381.583,A -85,B 0,C 180,E1 -17130.193,E2 -17130.193} C_VEL
LIN {X 0,Y 285.348,Z 372.61,A -85,B 0,C 180,E1 -17131.973,E2 -17131.973} C_VEL
LIN {X 0,Y 286.139,Z 362.094,A -85,B 0,C 180,E1 -17133.618,E2 -17133.618} C_VEL
LIN {X 0,Y 286.878,Z 351.313,A -85,B 0,C 180,E1 -17134.934,E2 -17134.934} C_VEL
LIN {X 0,Y 287.548,Z 339.484,A -85,B 0,C 180,E1 -17136.043,E2 -17136.043} C_VEL
LIN {X 0,Y 288.104,Z 327.303,A -85,B 0,C 180,E1 -17136.877,E2 -17136.877} C_VEL
LIN {X 0,Y 288.441,Z 313.861,A -85,B 0,C 180,E1 -17137.479,E2 -17137.479} C_VEL
LIN {X 0,Y 290.006,Z 256.936,A -85,B 0,C 180,E1 -17139.396,E2 -17139.396} C_VEL
LIN {X 0,Y 286.793,Z 233.142,A -85,B 0,C 180,E1 -17140.421,E2 -17140.421} C_VEL
LIN {X 0,Y 287.266,Z 224.429,A -85,B 0,C 180,E1 -17142.78,E2 -17142.78} C_VEL
LIN {X 0,Y 285.406,Z 214.446,A -85,B 0,C 180,E1 -17145.753,E2 -17145.753} C_VEL
LIN {X 0,Y 284.335,Z 209.178,A -85,B 0,C 180,E1 -17147.438,E2 -17147.438} C_VEL
LIN {X 0,Y 284.311,Z 209.072,A -85,B 0,C 180,E1 -17151.83,E2 -17151.83} C_VEL
LIN {X 0,Y 284.308,Z 209.071,A -85,B 0,C 180,E1 -17155.35,E2 -17155.35} C_VEL
LIN {X 0,Y 284.295,Z 209.07,A -85,B 0,C 180,E1 -17158.725,E2 -17158.725} C_VEL
LIN {X 0,Y 284.396,Z 209.057,A -85,B 0,C 180,E1 -17162.825,E2 -17162.825} C_VEL
LIN {X 0,Y 284.365,Z 209.061,A -85,B 0,C 180,E1 -17166.706,E2 -17166.706} C_VEL
LIN {X 0,Y 284.403,Z 209.06,A -85,B 0,C 180,E1 -17171.261,E2 -17171.261} C_VEL
LIN {X 0,Y 284.49,Z 209.044,A -85,B 0,C 180,E1 -17174.458,E2 -17174.458} C_VEL
LIN {X 0,Y 284.487,Z 209.046,A -85,B 0,C 180,E1 -17178.601,E2 -17178.601} C_VEL
LIN {X 0,Y 284.657,Z 209.026,A -85,B 0,C 180,E1 -17181.48,E2 -17181.48} C_VEL
LIN {X 0,Y 284.6,Z 209.031,A -85,B 0,C 180,E1 -17184.33,E2 -17184.33} C_VEL
LIN {X 0,Y 284.853,Z 209,A -85,B 0,C 180,E1 -17188.585,E2 -17188.585} C_VEL
LIN {X 0,Y 284.853,Z 209.002,A -85,B 0,C 180,E1 -17191.413,E2 -17191.413} C_VEL
LIN {X 0,Y 284.69,Z 209.023,A -85,B 0,C 180,E1 -17197.089,E2 -17197.089} C_VEL
LIN {X 0,Y 284.563,Z 209.035,A -85,B 0,C 180,E1 -17199.954,E2 -17199.954} C_VEL
LIN {X 0,Y 284.478,Z 209.047,A -85,B 0,C 180,E1 -17204.302,E2 -17204.302} C_VEL
LIN {X 0,Y 284.421,Z 209.055,A -85,B 0,C 180,E1 -17207.247,E2 -17207.247} C_VEL
LIN {X 0,Y 284.374,Z 209.061,A -85,B 0,C 180,E1 -17210.241,E2 -17210.241} C_VEL
LIN {X 0,Y 284.364,Z 209.06,A -85,B 0,C 180,E1 -17213.875,E2 -17213.875} C_VEL
LIN {X 0,Y 284.394,Z 209.058,A -85,B 0,C 180,E1 -17217.174,E2 -17217.174} C_VEL
LIN {X 0,Y 284.29,Z 209.07,A -85,B 0,C 180,E1 -17221.273,E2 -17221.273} C_VEL
LIN {X 0,Y 284.356,Z 209.062,A -85,B 0,C 180,E1 -17225.353,E2 -17225.353} C_VEL
LIN {X 0,Y 284.331,Z 209.067,A -85,B 0,C 180,E1 -17228.164,E2 -17228.164} C_VEL
LIN {X 0,Y 284.335,Z 209.066,A -85,B 0,C 180,E1 -17232.14,E2 -17232.14} C_VEL
LIN {X 0,Y 284.311,Z 209.071,A -85,B 0,C 180,E1 -17236.201,E2 -17236.201} C_VEL
LIN {X 0,Y 284.344,Z 209.065,A -85,B 0,C 180,E1 -17240.013,E2 -17240.013} C_VEL
LIN {X 0,Y 284.348,Z 209.063,A -85,B 0,C 180,E1 -17243.617,E2 -17243.617} C_VEL
LIN {X 0,Y 284.301,Z 209.068,A -85,B 0,C 180,E1 -17247.189,E2 -17247.189} C_VEL
LIN {X 0,Y 284.352,Z 209.065,A -85,B 0,C 180,E1 -17250.376,E2 -17250.376} C_VEL
LIN {X 0,Y 284.37,Z 209.061,A -85,B 0,C 180,E1 -17253.587,E2 -17253.587} C_VEL
LIN {X 0,Y 284.358,Z 209.061,A -85,B 0,C 180,E1 -17256.707,E2 -17256.707} C_VEL
LIN {X 0,Y 284.396,Z 209.057,A -85,B 0,C 180,E1 -17261.262,E2 -17261.262} C_VEL
LIN {X 0,Y 284.48,Z 209.046,A -85,B 0,C 180,E1 -17264.546,E2 -17264.546} C_VEL
LIN {X 0,Y 284.48,Z 209.047,A -85,B 0,C 180,E1 -17268.602,E2 -17268.602} C_VEL
LIN {X 0,Y 284.579,Z 209.034,A -85,B 0,C 180,E1 -17270.7,E2 -17270.7} C_VEL
LIN {X 0,Y 283.99,Z 209.111,A -85,B 0,C 180,E1 -17271.881,E2 -17271.881} C_VEL
LIN {X 0,Y 281.063,Z 209.475,A -85,B 0,C 180,E1 -17273.801,E2 -17273.801} C_VEL
LIN {X 0,Y 278.606,Z 209.779,A -85,B 0,C 180,E1 -17275.363,E2 -17275.363} C_VEL
LIN {X 0,Y 277.673,Z 209.894,A -85,B 0,C 180,E1 -17276.575,E2 -17276.575} C_VEL
LIN {X 0,Y 277.666,Z 209.895,A -85,B 0,C 180,E1 -17276.985,E2 -17276.985} C_VEL
LIN {X 0,Y 277.875,Z 209.871,A -85,B 0,C 180,E1 -17280.001,E2 -17280.001} C_VEL
LIN {X 0,Y 277.691,Z 209.891,A -85,B 0,C 180,E1 -17282.902,E2 -17282.902} C_VEL
LIN {X 0,Y 277.646,Z 209.9,A -85,B 0,C 180,E1 -17287.272,E2 -17287.272} C_VEL
LIN {X 0,Y 277.5,Z 209.915,A -85,B 0,C 180,E1 -17290.212,E2 -17290.212} C_VEL
LIN {X 0,Y 277.429,Z 209.925,A -85,B 0,C 180,E1 -17294.675,E2 -17294.675} C_VEL
LIN {X 0,Y 277.339,Z 209.938,A -85,B 0,C 180,E1 -17299.235,E2 -17299.235} C_VEL
LIN {X 0,Y 277.313,Z 209.939,A -85,B 0,C 180,E1 -17304.171,E2 -17304.171} C_VEL
LIN {X 0,Y 277.318,Z 209.941,A -85,B 0,C 180,E1 -17307.505,E2 -17307.505} C_VEL
LIN {X 0,Y 277.268,Z 209.945,A -85,B 0,C 180,E1 -17310.483,E2 -17310.483} C_VEL
LIN {X 0,Y 277.243,Z 209.948,A -85,B 0,C 180,E1 -17313.897,E2 -17313.897} C_VEL
LIN {X 0,Y 277.261,Z 209.948,A -85,B 0,C 180,E1 -17317.471,E2 -17317.471} C_VEL
LIN {X 0,Y 277.206,Z 209.956,A -85,B 0,C 180,E1 -17321.238,E2 -17321.238} C_VEL
LIN {X 0,Y 277.198,Z 209.957,A -85,B 0,C 180,E1 -17325.228,E2 -17325.228} C_VEL
LIN {X 0,Y 277.22,Z 209.953,A -85,B 0,C 180,E1 -17329.514,E2 -17329.514} C_VEL
LIN {X 0,Y 277.266,Z 209.949,A -85,B 0,C 180,E1 -17332.532,E2 -17332.532} C_VEL
LIN {X 0,Y 277.339,Z 210.189,A -85,B 0,C 180,E1 -17334.262,E2 -17334.262} C_VEL
LIN {X 0,Y 280.715,Z 225.337,A -85,B 0,C 180,E1 -17338.282,E2 -17338.282} C_VEL
LIN {X 0,Y 283.422,Z 238.077,A -85,B 0,C 180,E1 -17341.495,E2 -17341.495} C_VEL
LIN {X 0,Y 280.788,Z 257.095,A -85,B 0,C 180,E1 -17345.805,E2 -17345.805} C_VEL
LIN {X 0,Y 280.701,Z 258.52,A -85,B 0,C 180,E1 -17345.994,E2 -17345.994} C_VEL
LIN {X 0,Y 283.207,Z 292.723,A -85,B 0,C 180,E1 -17347.242,E2 -17347.242} C_VEL
LIN {X 0,Y 283.589,Z 299.646,A -85,B 0,C 180,E1 -17347.484,E2 -17347.484} C_VEL
LIN {X 0,Y 282.013,Z 361.675,A -85,B 0,C 180,E1 -17349.439,E2 -17349.439} C_VEL
LIN {X 0,Y 281.302,Z 374.286,A -85,B 0,C 180,E1 -17350.1,E2 -17350.1} C_VEL
LIN {X 0,Y 280.445,Z 386.099,A -85,B 0,C 180,E1 -17350.988,E2 -17350.988} C_VEL
LIN {X 0,Y 279.428,Z 398.435,A -85,B 0,C 180,E1 -17352.245,E2 -17352.245} C_VEL
LIN {X 0,Y 278.431,Z 409.373,A -85,B 0,C 180,E1 -17353.681,E2 -17353.681} C_VEL
LIN {X 0,Y 277.44,Z 419.309,A -85,B 0,C 180,E1 -17355.327,E2 -17355.327} C_VEL
LIN {X 0,Y 276.74,Z 428.277,A -85,B 0,C 180,E1 -17357.162,E2 -17357.162} C_VEL
LIN {X 0,Y 276.163,Z 436.846,A -85,B 0,C 180,E1 -17359.369,E2 -17359.369} C_VEL
LIN {X 0,Y 275.957,Z 443.643,A -85,B 0,C 180,E1 -17361.58,E2 -17361.58} C_VEL
LIN {X 0,Y 275.974,Z 447.883,A -85,B 0,C 180,E1 -17363.311,E2 -17363.311} C_VEL
LIN {X 0,Y 276.073,Z 452.299,A -85,B 0,C 180,E1 -17365.621,E2 -17365.621} C_VEL
LIN {X 0,Y 276.17,Z 454.385,A -85,B 0,C 180,E1 -17367.084,E2 -17367.084} C_VEL
LIN {X 0,Y 276.325,Z 455.97,A -85,B 0,C 180,E1 -17368.544,E2 -17368.544} C_VEL
LIN {X 0,Y 276.303,Z 457.078,A -85,B 0,C 180,E1 -17370.001,E2 -17370.001} C_VEL
LIN {X 0,Y 276.262,Z 457.68,A -85,B 0,C 180,E1 -17371.459,E2 -17371.459} C_VEL
LIN {X 0,Y 275.967,Z 457.81,A -85,B 0,C 180,E1 -17372.921,E2 -17372.921} C_VEL
LIN {X 0,Y 275.699,Z 457.52,A -85,B 0,C 180,E1 -17374.387,E2 -17374.387} C_VEL
LIN {X 0,Y 275.61,Z 456.68,A -85,B 0,C 180,E1 -17376.011,E2 -17376.011} C_VEL
LIN {X 0,Y 275.679,Z 454.038,A -85,B 0,C 180,E1 -17378.799,E2 -17378.799} C_VEL
LIN {X 0,Y 276.024,Z 450.806,A -85,B 0,C 180,E1 -17381.01,E2 -17381.01} C_VEL
LIN {X 0,Y 276.954,Z 446.516,A -85,B 0,C 180,E1 -17383.203,E2 -17383.203} C_VEL
LIN {X 0,Y 278.486,Z 440.026,A -85,B 0,C 180,E1 -17385.742,E2 -17385.742} C_VEL
LIN {X 0,Y 280.32,Z 432.992,A -85,B 0,C 180,E1 -17387.887,E2 -17387.887} C_VEL
LIN {X 0,Y 282.124,Z 425.863,A -85,B 0,C 180,E1 -17389.652,E2 -17389.652} C_VEL
LIN {X 0,Y 284.446,Z 417.294,A -85,B 0,C 180,E1 -17391.374,E2 -17391.374} C_VEL
LIN {X 0,Y 287.299,Z 405.668,A -85,B 0,C 180,E1 -17393.233,E2 -17393.233} C_VEL
LIN {X 0,Y 289.704,Z 395.147,A -85,B 0,C 180,E1 -17394.548,E2 -17394.548} C_VEL
LIN {X 0,Y 292.012,Z 383.522,A -85,B 0,C 180,E1 -17395.673,E2 -17395.673} C_VEL
LIN {X 0,Y 294.147,Z 370.458,A -85,B 0,C 180,E1 -17396.616,E2 -17396.616} C_VEL
LIN {X 0,Y 295.755,Z 356.328,A -85,B 0,C 180,E1 -17397.318,E2 -17397.318} C_VEL
LIN {X 0,Y 299.27,Z 301.687,A -85,B 0,C 180,E1 -17399.146,E2 -17399.146} C_VEL
LIN {X 0,Y 298.165,Z 286.16,A -85,B 0,C 180,E1 -17400.048,E2 -17400.048} C_VEL
LIN {X 0,Y 296.078,Z 269.81,A -85,B 0,C 180,E1 -17401.21,E2 -17401.21} C_VEL
LIN {X 0,Y 294.032,Z 258.237,A -85,B 0,C 180,E1 -17402.205,E2 -17402.205} C_VEL
LIN {X 0,Y 291.695,Z 253.076,A -85,B 0,C 180,E1 -17403.02,E2 -17403.02} C_VEL
LIN {X 0,Y 290.179,Z 245.603,A -85,B 0,C 180,E1 -17405.541,E2 -17405.541} C_VEL
LIN {X 0,Y 288.482,Z 239.02,A -85,B 0,C 180,E1 -17408.117,E2 -17408.117} C_VEL
LIN {X 0,Y 286.752,Z 233.694,A -85,B 0,C 180,E1 -17410.554,E2 -17410.554} C_VEL
LIN {X 0,Y 284.412,Z 227.023,A -85,B 0,C 180,E1 -17414.224,E2 -17414.224} C_VEL
LIN {X 0,Y 282.455,Z 222.139,A -85,B 0,C 180,E1 -17417.792,E2 -17417.792} C_VEL
LIN {X 0,Y 281.071,Z 218.755,A -85,B 0,C 180,E1 -17421.309,E2 -17421.309} C_VEL
LIN {X 0,Y 280.519,Z 217.425,A -85,B 0,C 180,E1 -17423.295,E2 -17423.295} C_VEL
LIN {X 0,Y 279.891,Z 216.328,A -85,B 0,C 180,E1 -17426.466,E2 -17426.466} C_VEL
LIN {X 0,Y 279.839,Z 216.216,A -85,B 0,C 180,E1 -17429.848,E2 -17429.848} C_VEL
LIN {X 0,Y 280.473,Z 217.169,A -85,B 0,C 180,E1 -17433.189,E2 -17433.189} C_VEL
LIN {X 0,Y 280.87,Z 218.128,A -85,B 0,C 180,E1 -17434.825,E2 -17434.825} C_VEL
LIN {X 0,Y 281.94,Z 220.896,A -85,B 0,C 180,E1 -17438.042,E2 -17438.042} C_VEL
LIN {X 0,Y 283.458,Z 224.588,A -85,B 0,C 180,E1 -17441.196,E2 -17441.196} C_VEL
LIN {X 0,Y 285.163,Z 229.238,A -85,B 0,C 180,E1 -17444.27,E2 -17444.27} C_VEL
LIN {X 0,Y 286.93,Z 234.794,A -85,B 0,C 180,E1 -17447.264,E2 -17447.264} C_VEL
LIN {X 0,Y 288.181,Z 238.966,A -85,B 0,C 180,E1 -17449.127,E2 -17449.127} C_VEL
LIN {X 0,Y 291.615,Z 244.692,A -85,B 0,C 180,E1 -17450.31,E2 -17450.31} C_VEL
LIN {X 0,Y 295.579,Z 252.012,A -85,B 0,C 180,E1 -17451.584,E2 -17451.584} C_VEL
LIN {X 0,Y 298.421,Z 258.09,A -85,B 0,C 180,E1 -17452.493,E2 -17452.493} C_VEL
LIN {X 0,Y 300.709,Z 270.317,A -85,B 0,C 180,E1 -17453.559,E2 -17453.559} C_VEL
LIN {X 0,Y 296.356,Z 325.146,A -85,B 0,C 180,E1 -17455.675,E2 -17455.675} C_VEL
LIN {X 0,Y 295.209,Z 337.681,A -85,B 0,C 180,E1 -17456.416,E2 -17456.416} C_VEL
LIN {X 0,Y 293.628,Z 349.968,A -85,B 0,C 180,E1 -17457.427,E2 -17457.427} C_VEL
LIN {X 0,Y 291.846,Z 360.856,A -85,B 0,C 180,E1 -17458.619,E2 -17458.619} C_VEL
LIN {X 0,Y 289.849,Z 370.701,A -85,B 0,C 180,E1 -17459.999,E2 -17459.999} C_VEL
LIN {X 0,Y 287.944,Z 378.725,A -85,B 0,C 180,E1 -17461.398,E2 -17461.398} C_VEL
LIN {X 0,Y 285.813,Z 386.782,A -85,B 0,C 180,E1 -17463.171,E2 -17463.171} C_VEL
LIN {X 0,Y 283.889,Z 393.317,A -85,B 0,C 180,E1 -17464.97,E2 -17464.97} C_VEL
LIN {X 0,Y 281.861,Z 399.407,A -85,B 0,C 180,E1 -17467.161,E2 -17467.161} C_VEL
LIN {X 0,Y 280.151,Z 403.911,A -85,B 0,C 180,E1 -17469.384,E2 -17469.384} C_VEL
LIN {X 0,Y 278.785,Z 406.984,A -85,B 0,C 180,E1 -17471.634,E2 -17471.634} C_VEL
LIN {X 0,Y 278.01,Z 408.312,A -85,B 0,C 180,E1 -17473.15,E2 -17473.15} C_VEL
LIN {X 0,Y 277.097,Z 409.247,A -85,B 0,C 180,E1 -17475.464,E2 -17475.464} C_VEL
LIN {X 0,Y 276.458,Z 408.914,A -85,B 0,C 180,E1 -17477.761,E2 -17477.761} C_VEL
LIN {X 0,Y 276.153,Z 407.656,A -85,B 0,C 180,E1 -17479.67,E2 -17479.67} C_VEL
LIN {X 0,Y 276.013,Z 405.382,A -85,B 0,C 180,E1 -17481.666,E2 -17481.666} C_VEL
LIN {X 0,Y 276.215,Z 401.366,A -85,B 0,C 180,E1 -17484.022,E2 -17484.022} C_VEL
LIN {X 0,Y 276.564,Z 395.666,A -85,B 0,C 180,E1 -17486.404,E2 -17486.404} C_VEL
LIN {X 0,Y 276.989,Z 389.547,A -85,B 0,C 180,E1 -17488.365,E2 -17488.365} C_VEL
LIN {X 0,Y 277.592,Z 381.343,A -85,B 0,C 180,E1 -17490.42,E2 -17490.42} C_VEL
LIN {X 0,Y 278.339,Z 372.174,A -85,B 0,C 180,E1 -17492.235,E2 -17492.235} C_VEL
LIN {X 0,Y 279.109,Z 362.218,A -85,B 0,C 180,E1 -17493.803,E2 -17493.803} C_VEL
LIN {X 0,Y 279.937,Z 350.241,A -85,B 0,C 180,E1 -17495.269,E2 -17495.269} C_VEL
LIN {X 0,Y 280.634,Z 338.1,A -85,B 0,C 180,E1 -17496.384,E2 -17496.384} C_VEL
LIN {X 0,Y 281.178,Z 324.78,A -85,B 0,C 180,E1 -17497.253,E2 -17497.253} C_VEL
LIN {X 0,Y 281.492,Z 309.29,A -85,B 0,C 180,E1 -17497.881,E2 -17497.881} C_VEL
LIN {X 0,Y 283.048,Z 257.693,A -85,B 0,C 180,E1 -17499.67,E2 -17499.67} C_VEL
LIN {X 0,Y 279.872,Z 233.637,A -85,B 0,C 180,E1 -17500.724,E2 -17500.724} C_VEL
LIN {X 0,Y 280.295,Z 226.642,A -85,B 0,C 180,E1 -17502.607,E2 -17502.607} C_VEL
LIN {X 0,Y 279.567,Z 221.347,A -85,B 0,C 180,E1 -17504.179,E2 -17504.179} C_VEL
LIN {X 0,Y 277.304,Z 210.113,A -85,B 0,C 180,E1 -17507.708,E2 -17507.708} C_VEL
LIN {X 0,Y 277.267,Z 209.946,A -85,B 0,C 180,E1 -17512.53,E2 -17512.53} C_VEL
LIN {X 0,Y 277.246,Z 209.949,A -85,B 0,C 180,E1 -17516.103,E2 -17516.103} C_VEL
LIN {X 0,Y 277.26,Z 209.95,A -85,B 0,C 180,E1 -17519.538,E2 -17519.538} C_VEL
LIN {X 0,Y 277.358,Z 209.934,A -85,B 0,C 180,E1 -17522.863,E2 -17522.863} C_VEL
LIN {X 0,Y 277.328,Z 209.938,A -85,B 0,C 180,E1 -17526.079,E2 -17526.079} C_VEL
LIN {X 0,Y 277.344,Z 209.936,A -85,B 0,C 180,E1 -17530.765,E2 -17530.765} C_VEL
LIN {X 0,Y 277.433,Z 209.929,A -85,B 0,C 180,E1 -17535.325,E2 -17535.325} C_VEL
LIN {X 0,Y 277.505,Z 209.915,A -85,B 0,C 180,E1 -17539.788,E2 -17539.788} C_VEL
LIN {X 0,Y 277.651,Z 209.897,A -85,B 0,C 180,E1 -17542.728,E2 -17542.728} C_VEL
LIN {X 0,Y 277.819,Z 209.876,A -85,B 0,C 180,E1 -17548.549,E2 -17548.549} C_VEL
LIN {X 0,Y 277.819,Z 209.878,A -85,B 0,C 180,E1 -17551.449,E2 -17551.449} C_VEL
LIN {X 0,Y 277.646,Z 209.899,A -85,B 0,C 180,E1 -17557.27,E2 -17557.27} C_VEL
LIN {X 0,Y 277.503,Z 209.915,A -85,B 0,C 180,E1 -17560.21,E2 -17560.21} C_VEL
LIN {X 0,Y 277.43,Z 209.928,A -85,B 0,C 180,E1 -17564.673,E2 -17564.673} C_VEL
LIN {X 0,Y 277.341,Z 209.937,A -85,B 0,C 180,E1 -17569.233,E2 -17569.233} C_VEL
LIN {X 0,Y 277.314,Z 209.939,A -85,B 0,C 180,E1 -17574.17,E2 -17574.17} C_VEL
LIN {X 0,Y 277.322,Z 209.938,A -85,B 0,C 180,E1 -17577.505,E2 -17577.505} C_VEL
LIN {X 0,Y 277.266,Z 209.949,A -85,B 0,C 180,E1 -17580.481,E2 -17580.481} C_VEL
LIN {X 0,Y 277.248,Z 209.946,A -85,B 0,C 180,E1 -17583.894,E2 -17583.894} C_VEL
LIN {X 0,Y 277.284,Z 209.943,A -85,B 0,C 180,E1 -17587.465,E2 -17587.465} C_VEL
LIN {X 0,Y 277.258,Z 209.945,A -85,B 0,C 180,E1 -17591.226,E2 -17591.226} C_VEL
LIN {X 0,Y 277.243,Z 209.948,A -85,B 0,C 180,E1 -17595.216,E2 -17595.216} C_VEL
LIN {X 0,Y 277.255,Z 209.945,A -85,B 0,C 180,E1 -17599.502,E2 -17599.502} C_VEL
LIN {X 0,Y 277.282,Z 209.946,A -85,B 0,C 180,E1 -17602.534,E2 -17602.534} C_VEL
LIN {X 0,Y 277.247,Z 209.951,A -85,B 0,C 180,E1 -17606.105,E2 -17606.105} C_VEL
LIN {X 0,Y 277.254,Z 209.946,A -85,B 0,C 180,E1 -17609.538,E2 -17609.538} C_VEL
LIN {X 0,Y 277.351,Z 209.935,A -85,B 0,C 180,E1 -17612.864,E2 -17612.864} C_VEL
LIN {X 0,Y 277.321,Z 209.941,A -85,B 0,C 180,E1 -17616.08,E2 -17616.08} C_VEL
LIN {X 0,Y 277.337,Z 209.936,A -85,B 0,C 180,E1 -17620.766,E2 -17620.766} C_VEL
LIN {X 0,Y 277.427,Z 209.924,A -85,B 0,C 180,E1 -17625.326,E2 -17625.326} C_VEL
LIN {X 0,Y 277.454,Z 209.926,A -85,B 0,C 180,E1 -17629.787,E2 -17629.787} C_VEL
LIN {X 0,Y 277.634,Z 209.898,A -85,B 0,C 180,E1 -17632.729,E2 -17632.729} C_VEL
LIN {X 0,Y 277.666,Z 209.895,A -85,B 0,C 180,E1 -17636.985,E2 -17636.985} C_VEL
LIN {X 0,Y 277.196,Z 209.958,A -85,B 0,C 180,E1 -17638.197,E2 -17638.197} C_VEL
LIN {X 0,Y 275.701,Z 210.146,A -85,B 0,C 180,E1 -17639.388,E2 -17639.388} C_VEL
LIN {X 0,Y 271.884,Z 210.618,A -85,B 0,C 180,E1 -17641.776,E2 -17641.776} C_VEL
LIN {X 0,Y 270.686,Z 210.764,A -85,B 0,C 180,E1 -17643.02,E2 -17643.02} C_VEL
LIN {X 0,Y 270.538,Z 210.78,A -85,B 0,C 180,E1 -17643.443,E2 -17643.443} C_VEL
LIN {X 0,Y 270.604,Z 210.779,A -85,B 0,C 180,E1 -17647.462,E2 -17647.462} C_VEL
LIN {X 0,Y 270.435,Z 210.794,A -85,B 0,C 180,E1 -17650.482,E2 -17650.482} C_VEL
LIN {X 0,Y 270.397,Z 210.803,A -85,B 0,C 180,E1 -17655.066,E2 -17655.066} C_VEL
LIN {X 0,Y 270.296,Z 210.814,A -85,B 0,C 180,E1 -17659.757,E2 -17659.757} C_VEL
LIN {X 0,Y 270.269,Z 210.817,A -85,B 0,C 180,E1 -17664.587,E2 -17664.587} C_VEL
LIN {X 0,Y 270.265,Z 210.817,A -85,B 0,C 180,E1 -17667.91,E2 -17667.91} C_VEL
LIN {X 0,Y 270.18,Z 210.831,A -85,B 0,C 180,E1 -17671.35,E2 -17671.35} C_VEL
LIN {X 0,Y 270.197,Z 210.829,A -85,B 0,C 180,E1 -17674.907,E2 -17674.907} C_VEL
LIN {X 0,Y 270.194,Z 210.828,A -85,B 0,C 180,E1 -17678.712,E2 -17678.712} C_VEL
LIN {X 0,Y 270.168,Z 210.831,A -85,B 0,C 180,E1 -17682.56,E2 -17682.56} C_VEL
LIN {X 0,Y 270.162,Z 210.834,A -85,B 0,C 180,E1 -17686.753,E2 -17686.753} C_VEL
LIN {X 0,Y 270.172,Z 210.831,A -85,B 0,C 180,E1 -17689.436,E2 -17689.436} C_VEL
LIN {X 0,Y 270.253,Z 210.943,A -85,B 0,C 180,E1 -17693.811,E2 -17693.811} C_VEL
LIN {X 0,Y 273.363,Z 224.753,A -85,B 0,C 180,E1 -17697.622,E2 -17697.622} C_VEL
LIN {X 0,Y 276.283,Z 238.122,A -85,B 0,C 180,E1 -17701.099,E2 -17701.099} C_VEL
LIN {X 0,Y 276.098,Z 241.516,A -85,B 0,C 180,E1 -17701.908,E2 -17701.908} C_VEL
LIN {X 0,Y 273.779,Z 257.549,A -85,B 0,C 180,E1 -17705.6,E2 -17705.6} C_VEL
LIN {X 0,Y 275.277,Z 282.02,A -85,B 0,C 180,E1 -17706.55,E2 -17706.55} C_VEL
LIN {X 0,Y 276.661,Z 298.289,A -85,B 0,C 180,E1 -17707.158,E2 -17707.158} C_VEL
LIN {X 0,Y 275.037,Z 360.864,A -85,B 0,C 180,E1 -17709.187,E2 -17709.187} C_VEL
LIN {X 0,Y 274.325,Z 373.539,A -85,B 0,C 180,E1 -17709.865,E2 -17709.865} C_VEL
LIN {X 0,Y 273.472,Z 385.417,A -85,B 0,C 180,E1 -17710.777,E2 -17710.777} C_VEL
LIN {X 0,Y 272.48,Z 396.974,A -85,B 0,C 180,E1 -17711.971,E2 -17711.971} C_VEL
LIN {X 0,Y 271.456,Z 408.186,A -85,B 0,C 180,E1 -17713.455,E2 -17713.455} C_VEL
LIN {X 0,Y 270.515,Z 417.175,A -85,B 0,C 180,E1 -17714.943,E2 -17714.943} C_VEL
LIN {X 0,Y 269.772,Z 426.392,A -85,B 0,C 180,E1 -17716.825,E2 -17716.825} C_VEL
LIN {X 0,Y 269.249,Z 433.922,A -85,B 0,C 180,E1 -17718.712,E2 -17718.712} C_VEL
LIN {X 0,Y 268.953,Z 441.202,A -85,B 0,C 180,E1 -17720.981,E2 -17720.981} C_VEL
LIN {X 0,Y 268.931,Z 446.876,A -85,B 0,C 180,E1 -17723.249,E2 -17723.249} C_VEL
LIN {X 0,Y 269.026,Z 451.172,A -85,B 0,C 180,E1 -17725.506,E2 -17725.506} C_VEL
LIN {X 0,Y 269.113,Z 453.368,A -85,B 0,C 180,E1 -17727.007,E2 -17727.007} C_VEL
LIN {X 0,Y 269.281,Z 455.018,A -85,B 0,C 180,E1 -17728.506,E2 -17728.506} C_VEL
LIN {X 0,Y 269.264,Z 456.181,A -85,B 0,C 180,E1 -17730.001,E2 -17730.001} C_VEL
LIN {X 0,Y 269.211,Z 456.889,A -85,B 0,C 180,E1 -17731.497,E2 -17731.497} C_VEL
LIN {X 0,Y 268.884,Z 457.077,A -85,B 0,C 180,E1 -17732.998,E2 -17732.998} C_VEL
LIN {X 0,Y 268.626,Z 456.846,A -85,B 0,C 180,E1 -17734.503,E2 -17734.503} C_VEL
LIN {X 0,Y 268.543,Z 456.211,A -85,B 0,C 180,E1 -17736.01,E2 -17736.01} C_VEL
LIN {X 0,Y 268.517,Z 455.116,A -85,B 0,C 180,E1 -17737.521,E2 -17737.521} C_VEL
LIN {X 0,Y 268.619,Z 453.586,A -85,B 0,C 180,E1 -17739.033,E2 -17739.033} C_VEL
LIN {X 0,Y 269.007,Z 450.494,A -85,B 0,C 180,E1 -17741.301,E2 -17741.301} C_VEL
LIN {X 0,Y 270.007,Z 446.361,A -85,B 0,C 180,E1 -17743.549,E2 -17743.549} C_VEL
LIN {X 0,Y 271.659,Z 440.079,A -85,B 0,C 180,E1 -17746.148,E2 -17746.148} C_VEL
LIN {X 0,Y 273.564,Z 433.198,A -85,B 0,C 180,E1 -17748.344,E2 -17748.344} C_VEL
LIN {X 0,Y 275.913,Z 424.775,A -85,B 0,C 180,E1 -17750.503,E2 -17750.503} C_VEL
LIN {X 0,Y 278.399,Z 416.193,A -85,B 0,C 180,E1 -17752.252,E2 -17752.252} C_VEL
LIN {X 0,Y 281.152,Z 405.658,A -85,B 0,C 180,E1 -17753.967,E2 -17753.967} C_VEL
LIN {X 0,Y 283.674,Z 395.296,A -85,B 0,C 180,E1 -17755.301,E2 -17755.301} C_VEL
LIN {X 0,Y 286.079,Z 383.91,A -85,B 0,C 180,E1 -17756.441,E2 -17756.441} C_VEL
LIN {X 0,Y 288.315,Z 371.345,A -85,B 0,C 180,E1 -17757.394,E2 -17757.394} C_VEL
LIN {X 0,Y 290.045,Z 358.179,A -85,B 0,C 180,E1 -17758.099,E2 -17758.099} C_VEL
LIN {X 0,Y 291.728,Z 335.054,A -85,B 0,C 180,E1 -17758.919,E2 -17758.919} C_VEL
LIN {X 0,Y 293.912,Z 302.444,A -85,B 0,C 180,E1 -17760.043,E2 -17760.043} C_VEL
LIN {X 0,Y 292.964,Z 287.713,A -85,B 0,C 180,E1 -17760.931,E2 -17760.931} C_VEL
LIN {X 0,Y 290.84,Z 270.243,A -85,B 0,C 180,E1 -17762.246,E2 -17762.246} C_VEL
LIN {X 0,Y 289.372,Z 261.967,A -85,B 0,C 180,E1 -17763,E2 -17763} C_VEL
LIN {X 0,Y 286.063,Z 255.185,A -85,B 0,C 180,E1 -17764.152,E2 -17764.152} C_VEL
LIN {X 0,Y 284.85,Z 252.285,A -85,B 0,C 180,E1 -17764.699,E2 -17764.699} C_VEL
LIN {X 0,Y 283.228,Z 245.053,A -85,B 0,C 180,E1 -17767.434,E2 -17767.434} C_VEL
LIN {X 0,Y 281.588,Z 239.399,A -85,B 0,C 180,E1 -17769.967,E2 -17769.967} C_VEL
LIN {X 0,Y 279.585,Z 233.356,A -85,B 0,C 180,E1 -17773.198,E2 -17773.198} C_VEL
LIN {X 0,Y 278.162,Z 229.426,A -85,B 0,C 180,E1 -17775.778,E2 -17775.778} C_VEL
LIN {X 0,Y 276.785,Z 225.933,A -85,B 0,C 180,E1 -17778.686,E2 -17778.686} C_VEL
LIN {X 0,Y 275.551,Z 222.885,A -85,B 0,C 180,E1 -17782.256,E2 -17782.256} C_VEL
LIN {X 0,Y 274.82,Z 221.322,A -85,B 0,C 180,E1 -17785.763,E2 -17785.763} C_VEL
LIN {X 0,Y 274.611,Z 221.031,A -85,B 0,C 180,E1 -17789.212,E2 -17789.212} C_VEL
LIN {X 0,Y 275.275,Z 222.043,A -85,B 0,C 180,E1 -17793.328,E2 -17793.328} C_VEL
LIN {X 0,Y 276.01,Z 224.197,A -85,B 0,C 180,E1 -17796.444,E2 -17796.444} C_VEL
LIN {X 0,Y 277.303,Z 227.341,A -85,B 0,C 180,E1 -17799.675,E2 -17799.675} C_VEL
LIN {X 0,Y 278.999,Z 231.996,A -85,B 0,C 180,E1 -17803.182,E2 -17803.182} C_VEL
LIN {X 0,Y 280.647,Z 237.18,A -85,B 0,C 180,E1 -17806.237,E2 -17806.237} C_VEL
LIN {X 0,Y 281.488,Z 239.684,A -85,B 0,C 180,E1 -17807.418,E2 -17807.418} C_VEL
LIN {X 0,Y 287.242,Z 248.827,A -85,B 0,C 180,E1 -17809.541,E2 -17809.541} C_VEL
LIN {X 0,Y 291.5,Z 257.064,A -85,B 0,C 180,E1 -17811.019,E2 -17811.019} C_VEL
LIN {X 0,Y 293.751,Z 262.026,A -85,B 0,C 180,E1 -17811.773,E2 -17811.773} C_VEL
LIN {X 0,Y 295.442,Z 271.873,A -85,B 0,C 180,E1 -17812.673,E2 -17812.673} C_VEL
LIN {X 0,Y 290.942,Z 325.671,A -85,B 0,C 180,E1 -17814.791,E2 -17814.791} C_VEL
LIN {X 0,Y 289.655,Z 338.755,A -85,B 0,C 180,E1 -17815.575,E2 -17815.575} C_VEL
LIN {X 0,Y 288.139,Z 349.817,A -85,B 0,C 180,E1 -17816.503,E2 -17816.503} C_VEL
LIN {X 0,Y 286.173,Z 360.869,A -85,B 0,C 180,E1 -17817.712,E2 -17817.712} C_VEL
LIN {X 0,Y 283.833,Z 371.866,A -85,B 0,C 180,E1 -17819.29,E2 -17819.29} C_VEL
LIN {X 0,Y 281.686,Z 380.26,A -85,B 0,C 180,E1 -17820.804,E2 -17820.804} C_VEL
LIN {X 0,Y 279.512,Z 387.944,A -85,B 0,C 180,E1 -17822.548,E2 -17822.548} C_VEL
LIN {X 0,Y 277.495,Z 394.277,A -85,B 0,C 180,E1 -17824.357,E2 -17824.357} C_VEL
LIN {X 0,Y 275.3,Z 400.3,A -85,B 0,C 180,E1 -17826.603,E2 -17826.603} C_VEL
LIN {X 0,Y 273.478,Z 404.743,A -85,B 0,C 180,E1 -17828.869,E2 -17828.869} C_VEL
LIN {X 0,Y 272.084,Z 407.629,A -85,B 0,C 180,E1 -17831.021,E2 -17831.021} C_VEL
LIN {X 0,Y 270.801,Z 409.547,A -85,B 0,C 180,E1 -17833.507,E2 -17833.507} C_VEL
LIN {X 0,Y 269.983,Z 410.023,A -85,B 0,C 180,E1 -17835.6,E2 -17835.6} C_VEL
LIN {X 0,Y 269.281,Z 409.216,A -85,B 0,C 180,E1 -17838.251,E2 -17838.251} C_VEL
LIN {X 0,Y 269.06,Z 407.892,A -85,B 0,C 180,E1 -17839.89,E2 -17839.89} C_VEL
LIN {X 0,Y 268.963,Z 404.894,A -85,B 0,C 180,E1 -17842.264,E2 -17842.264} C_VEL
LIN {X 0,Y 269.195,Z 400.31,A -85,B 0,C 180,E1 -17844.69,E2 -17844.69} C_VEL
LIN {X 0,Y 269.46,Z 396.298,A -85,B 0,C 180,E1 -17846.32,E2 -17846.32} C_VEL
LIN {X 0,Y 269.898,Z 390.024,A -85,B 0,C 180,E1 -17848.373,E2 -17848.373} C_VEL
LIN {X 0,Y 270.47,Z 381.962,A -85,B 0,C 180,E1 -17850.443,E2 -17850.443} C_VEL
LIN {X 0,Y 271.251,Z 372.828,A -85,B 0,C 180,E1 -17852.301,E2 -17852.301} C_VEL
LIN {X 0,Y 272.06,Z 362.566,A -85,B 0,C 180,E1 -17853.96,E2 -17853.96} C_VEL
LIN {X 0,Y 272.879,Z 351.013,A -85,B 0,C 180,E1 -17855.414,E2 -17855.414} C_VEL
LIN {X 0,Y 273.623,Z 338.319,A -85,B 0,C 180,E1 -17856.608,E2 -17856.608} C_VEL
LIN {X 0,Y 274.204,Z 324.845,A -85,B 0,C 180,E1 -17857.499,E2 -17857.499} C_VEL
LIN {X 0,Y 274.605,Z 307.145,A -85,B 0,C 180,E1 -17858.215,E2 -17858.215} C_VEL
LIN {X 0,Y 276.144,Z 258.715,A -85,B 0,C 180,E1 -17859.941,E2 -17859.941} C_VEL
LIN {X 0,Y 272.903,Z 233.935,A -85,B 0,C 180,E1 -17861.055,E2 -17861.055} C_VEL
LIN {X 0,Y 273.307,Z 226.92,A -85,B 0,C 180,E1 -17862.987,E2 -17862.987} C_VEL
LIN {X 0,Y 271.366,Z 216.467,A -85,B 0,C 180,E1 -17866.225,E2 -17866.225} C_VEL
LIN {X 0,Y 270.229,Z 210.947,A -85,B 0,C 180,E1 -17868.076,E2 -17868.076} C_VEL
LIN {X 0,Y 270.206,Z 210.828,A -85,B 0,C 180,E1 -17871.373,E2 -17871.373} C_VEL
LIN {X 0,Y 270.201,Z 210.827,A -85,B 0,C 180,E1 -17875.094,E2 -17875.094} C_VEL
LIN {X 0,Y 270.199,Z 210.827,A -85,B 0,C 180,E1 -17879.13,E2 -17879.13} C_VEL
LIN {X 0,Y 270.264,Z 210.818,A -85,B 0,C 180,E1 -17882.145,E2 -17882.145} C_VEL
LIN {X 0,Y 270.276,Z 210.82,A -85,B 0,C 180,E1 -17885.518,E2 -17885.518} C_VEL
LIN {X 0,Y 270.3,Z 210.813,A -85,B 0,C 180,E1 -17890.243,E2 -17890.243} C_VEL
LIN {X 0,Y 270.401,Z 210.801,A -85,B 0,C 180,E1 -17894.934,E2 -17894.934} C_VEL
LIN {X 0,Y 270.44,Z 210.797,A -85,B 0,C 180,E1 -17899.518,E2 -17899.518} C_VEL
LIN {X 0,Y 270.609,Z 210.774,A -85,B 0,C 180,E1 -17902.538,E2 -17902.538} C_VEL
LIN {X 0,Y 270.785,Z 210.752,A -85,B 0,C 180,E1 -17908.512,E2 -17908.512} C_VEL
LIN {X 0,Y 270.785,Z 210.754,A -85,B 0,C 180,E1 -17911.486,E2 -17911.486} C_VEL
LIN {X 0,Y 270.604,Z 210.774,A -85,B 0,C 180,E1 -17917.46,E2 -17917.46} C_VEL
LIN {X 0,Y 270.438,Z 210.797,A -85,B 0,C 180,E1 -17920.48,E2 -17920.48} C_VEL
LIN {X 0,Y 270.399,Z 210.802,A -85,B 0,C 180,E1 -17925.064,E2 -17925.064} C_VEL
LIN {X 0,Y 270.297,Z 210.813,A -85,B 0,C 180,E1 -17929.755,E2 -17929.755} C_VEL
LIN {X 0,Y 270.269,Z 210.819,A -85,B 0,C 180,E1 -17934.585,E2 -17934.585} C_VEL
LIN {X 0,Y 270.267,Z 210.817,A -85,B 0,C 180,E1 -17937.908,E2 -17937.908} C_VEL
LIN {X 0,Y 270.178,Z 210.827,A -85,B 0,C 180,E1 -17941.347,E2 -17941.347} C_VEL
LIN {X 0,Y 270.21,Z 210.826,A -85,B 0,C 180,E1 -17944.903,E2 -17944.903} C_VEL
LIN {X 0,Y 270.216,Z 210.826,A -85,B 0,C 180,E1 -17948.716,E2 -17948.716} C_VEL
LIN {X 0,Y 270.216,Z 210.826,A -85,B 0,C 180,E1 -17952.548,E2 -17952.548} C_VEL
LIN {X 0,Y 270.197,Z 210.827,A -85,B 0,C 180,E1 -17956.742,E2 -17956.742} C_VEL
LIN {X 0,Y 270.206,Z 210.823,A -85,B 0,C 180,E1 -17959.441,E2 -17959.441} C_VEL
LIN {X 0,Y 270.25,Z 210.82,A -85,B 0,C 180,E1 -17963.721,E2 -17963.721} C_VEL
LIN {X 0,Y 270.197,Z 210.825,A -85,B 0,C 180,E1 -17966.893,E2 -17966.893} C_VEL
LIN {X 0,Y 270.213,Z 210.826,A -85,B 0,C 180,E1 -17970.386,E2 -17970.386} C_VEL
LIN {X 0,Y 270.256,Z 210.82,A -85,B 0,C 180,E1 -17973.764,E2 -17973.764} C_VEL
LIN {X 0,Y 270.225,Z 210.82,A -85,B 0,C 180,E1 -17977.039,E2 -17977.039} C_VEL
LIN {X 0,Y 270.294,Z 210.816,A -85,B 0,C 180,E1 -17980.245,E2 -17980.245} C_VEL
LIN {X 0,Y 270.395,Z 210.799,A -85,B 0,C 180,E1 -17984.936,E2 -17984.936} C_VEL
LIN {X 0,Y 270.405,Z 210.802,A -85,B 0,C 180,E1 -17989.518,E2 -17989.518} C_VEL
LIN {X 0,Y 270.591,Z 210.776,A -85,B 0,C 180,E1 -17992.539,E2 -17992.539} C_VEL
LIN {X 0,Y 270.78,Z 210.753,A -85,B 0,C 180,E1 -17998.513,E2 -17998.513} C_VEL
LIN {X 0,Y 270.78,Z 210.756,A -85,B 0,C 180,E1 -18001.488,E2 -18001.488} C_VEL
LIN {X 0,Y 270.538,Z 210.78,A -85,B 0,C 180,E1 -18003.443,E2 -18003.443} C_VEL
LIN {X 0,Y 269.76,Z 210.881,A -85,B 0,C 180,E1 -18004.686,E2 -18004.686} C_VEL
LIN {X 0,Y 266.949,Z 211.23,A -85,B 0,C 180,E1 -18006.716,E2 -18006.716} C_VEL
LIN {X 0,Y 263.792,Z 211.625,A -85,B 0,C 180,E1 -18009.211,E2 -18009.211} C_VEL
LIN {X 0,Y 263.424,Z 211.667,A -85,B 0,C 180,E1 -18010.072,E2 -18010.072} C_VEL
LIN {X 0,Y 263.302,Z 211.686,A -85,B 0,C 180,E1 -18013.901,E2 -18013.901} C_VEL
LIN {X 0,Y 263.265,Z 211.691,A -85,B 0,C 180,E1 -18017.077,E2 -18017.077} C_VEL
LIN {X 0,Y 263.212,Z 211.696,A -85,B 0,C 180,E1 -18020.852,E2 -18020.852} C_VEL
LIN {X 0,Y 263.203,Z 211.7,A -85,B 0,C 180,E1 -18025.293,E2 -18025.293} C_VEL
LIN {X 0,Y 263.161,Z 211.703,A -85,B 0,C 180,E1 -18028.733,E2 -18028.733} C_VEL
LIN {X 0,Y 263.128,Z 211.706,A -85,B 0,C 180,E1 -18032.29,E2 -18032.29} C_VEL
LIN {X 0,Y 263.178,Z 211.702,A -85,B 0,C 180,E1 -18036.764,E2 -18036.764} C_VEL
LIN {X 0,Y 263.121,Z 211.708,A -85,B 0,C 180,E1 -18041.595,E2 -18041.595} C_VEL
LIN {X 0,Y 263.102,Z 211.71,A -85,B 0,C 180,E1 -18046.157,E2 -18046.157} C_VEL
LIN {X 0,Y 263.104,Z 211.711,A -85,B 0,C 180,E1 -18050.129,E2 -18050.129} C_VEL
LIN {X 0,Y 263.223,Z 211.93,A -85,B 0,C 180,E1 -18053.476,E2 -18053.476} C_VEL
LIN {X 0,Y 266.49,Z 226.455,A -85,B 0,C 180,E1 -18057.557,E2 -18057.557} C_VEL
LIN {X 0,Y 269.334,Z 239.924,A -85,B 0,C 180,E1 -18061.137,E2 -18061.137} C_VEL
LIN {X 0,Y 267.613,Z 251.504,A -85,B 0,C 180,E1 -18063.905,E2 -18063.905} C_VEL
LIN {X 0,Y 266.851,Z 257.159,A -85,B 0,C 180,E1 -18065.244,E2 -18065.244} C_VEL
LIN {X 0,Y 268.254,Z 281.486,A -85,B 0,C 180,E1 -18066.208,E2 -18066.208} C_VEL
LIN {X 0,Y 269.687,Z 299.351,A -85,B 0,C 180,E1 -18066.896,E2 -18066.896} C_VEL
LIN {X 0,Y 268.023,Z 360.911,A -85,B 0,C 180,E1 -18068.968,E2 -18068.968} C_VEL
LIN {X 0,Y 267.251,Z 374.053,A -85,B 0,C 180,E1 -18069.71,E2 -18069.71} C_VEL
LIN {X 0,Y 266.305,Z 386.524,A -85,B 0,C 180,E1 -18070.74,E2 -18070.74} C_VEL
LIN {X 0,Y 265.284,Z 398.533,A -85,B 0,C 180,E1 -18072.065,E2 -18072.065} C_VEL
LIN {X 0,Y 264.273,Z 409.118,A -85,B 0,C 180,E1 -18073.573,E2 -18073.573} C_VEL
LIN {X 0,Y 263.279,Z 418.9,A -85,B 0,C 180,E1 -18075.311,E2 -18075.311} C_VEL
LIN {X 0,Y 262.568,Z 427.702,A -85,B 0,C 180,E1 -18077.244,E2 -18077.244} C_VEL
LIN {X 0,Y 262.018,Z 436.108,A -85,B 0,C 180,E1 -18079.57,E2 -18079.57} C_VEL
LIN {X 0,Y 261.86,Z 441.762,A -85,B 0,C 180,E1 -18081.513,E2 -18081.513} C_VEL
LIN {X 0,Y 261.907,Z 447.169,A -85,B 0,C 180,E1 -18083.839,E2 -18083.839} C_VEL
LIN {X 0,Y 262.009,Z 451.211,A -85,B 0,C 180,E1 -18086.156,E2 -18086.156} C_VEL
LIN {X 0,Y 262.236,Z 454.044,A -85,B 0,C 180,E1 -18088.465,E2 -18088.465} C_VEL
LIN {X 0,Y 262.225,Z 455.271,A -85,B 0,C 180,E1 -18090.001,E2 -18090.001} C_VEL
LIN {X 0,Y 262.159,Z 456.048,A -85,B 0,C 180,E1 -18091.537,E2 -18091.537} C_VEL
LIN {X 0,Y 261.805,Z 456.344,A -85,B 0,C 180,E1 -18093.079,E2 -18093.079} C_VEL
LIN {X 0,Y 261.477,Z 455.673,A -85,B 0,C 180,E1 -18096.012,E2 -18096.012} C_VEL
LIN {X 0,Y 261.427,Z 454.609,A -85,B 0,C 180,E1 -18097.726,E2 -18097.726} C_VEL
LIN {X 0,Y 261.546,Z 453.166,A -85,B 0,C 180,E1 -18099.279,E2 -18099.279} C_VEL
LIN {X 0,Y 262.007,Z 450.206,A -85,B 0,C 180,E1 -18101.607,E2 -18101.607} C_VEL
LIN {X 0,Y 263.077,Z 446.205,A -85,B 0,C 180,E1 -18103.913,E2 -18103.913} C_VEL
LIN {X 0,Y 264.51,Z 441.068,A -85,B 0,C 180,E1 -18106.2,E2 -18106.2} C_VEL
LIN {X 0,Y 266.444,Z 434.695,A -85,B 0,C 180,E1 -18108.454,E2 -18108.454} C_VEL
LIN {X 0,Y 268.857,Z 426.817,A -85,B 0,C 180,E1 -18110.665,E2 -18110.665} C_VEL
LIN {X 0,Y 271.895,Z 416.961,A -85,B 0,C 180,E1 -18112.814,E2 -18112.814} C_VEL
LIN {X 0,Y 274.755,Z 406.841,A -85,B 0,C 180,E1 -18114.562,E2 -18114.562} C_VEL
LIN {X 0,Y 277.705,Z 395.578,A -85,B 0,C 180,E1 -18116.087,E2 -18116.087} C_VEL
LIN {X 0,Y 280.235,Z 384.647,A -85,B 0,C 180,E1 -18117.239,E2 -18117.239} C_VEL
LIN {X 0,Y 282.758,Z 371.336,A -85,B 0,C 180,E1 -18118.282,E2 -18118.282} C_VEL
LIN {X 0,Y 284.571,Z 358.555,A -85,B 0,C 180,E1 -18118.992,E2 -18118.992} C_VEL
LIN {X 0,Y 286.124,Z 338.9,A -85,B 0,C 180,E1 -18119.723,E2 -18119.723} C_VEL
LIN {X 0,Y 288.706,Z 303.795,A -85,B 0,C 180,E1 -18120.957,E2 -18120.957} C_VEL
LIN {X 0,Y 287.84,Z 288.488,A -85,B 0,C 180,E1 -18121.921,E2 -18121.921} C_VEL
LIN {X 0,Y 285.911,Z 271.845,A -85,B 0,C 180,E1 -18123.236,E2 -18123.236} C_VEL
LIN {X 0,Y 284.974,Z 265.971,A -85,B 0,C 180,E1 -18123.789,E2 -18123.789} C_VEL
LIN {X 0,Y 280.716,Z 257.001,A -85,B 0,C 180,E1 -18125.389,E2 -18125.389} C_VEL
LIN {X 0,Y 278.096,Z 251.756,A -85,B 0,C 180,E1 -18126.523,E2 -18126.523} C_VEL
LIN {X 0,Y 276.333,Z 244.865,A -85,B 0,C 180,E1 -18129.482,E2 -18129.482} C_VEL
LIN {X 0,Y 274.192,Z 238.203,A -85,B 0,C 180,E1 -18133.072,E2 -18133.072} C_VEL
LIN {X 0,Y 272.579,Z 233.556,A -85,B 0,C 180,E1 -18136.215,E2 -18136.215} C_VEL
LIN {X 0,Y 271.134,Z 229.803,A -85,B 0,C 180,E1 -18139.607,E2 -18139.607} C_VEL
LIN {X 0,Y 270.085,Z 227.191,A -85,B 0,C 180,E1 -18143.237,E2 -18143.237} C_VEL
LIN {X 0,Y 269.496,Z 226.043,A -85,B 0,C 180,E1 -18146.565,E2 -18146.565} C_VEL
LIN {X 0,Y 269.47,Z 225.991,A -85,B 0,C 180,E1 -18150.294,E2 -18150.294} C_VEL
LIN {X 0,Y 270.146,Z 227.068,A -85,B 0,C 180,E1 -18153.751,E2 -18153.751} C_VEL
LIN {X 0,Y 270.941,Z 229.49,A -85,B 0,C 180,E1 -18157.101,E2 -18157.101} C_VEL
LIN {X 0,Y 272.225,Z 232.812,A -85,B 0,C 180,E1 -18160.389,E2 -18160.389} C_VEL
LIN {X 0,Y 273.703,Z 237.164,A -85,B 0,C 180,E1 -18163.593,E2 -18163.593} C_VEL
LIN {X 0,Y 274.757,Z 240.309,A -85,B 0,C 180,E1 -18165.413,E2 -18165.413} C_VEL
LIN {X 0,Y 278.873,Z 246.664,A -85,B 0,C 180,E1 -18167.19,E2 -18167.19} C_VEL
LIN {X 0,Y 283.645,Z 254.456,A -85,B 0,C 180,E1 -18169.02,E2 -18169.02} C_VEL
LIN {X 0,Y 287.809,Z 262.869,A -85,B 0,C 180,E1 -18170.557,E2 -18170.557} C_VEL
LIN {X 0,Y 289.109,Z 266.052,A -85,B 0,C 180,E1 -18171.035,E2 -18171.035} C_VEL
LIN {X 0,Y 290.327,Z 273.949,A -85,B 0,C 180,E1 -18171.757,E2 -18171.757} C_VEL
LIN {X 0,Y 285.637,Z 326.158,A -85,B 0,C 180,E1 -18173.864,E2 -18173.864} C_VEL
LIN {X 0,Y 284.342,Z 338.363,A -85,B 0,C 180,E1 -18174.596,E2 -18174.596} C_VEL
LIN {X 0,Y 282.659,Z 350.265,A -85,B 0,C 180,E1 -18175.591,E2 -18175.591} C_VEL
LIN {X 0,Y 280.687,Z 360.96,A -85,B 0,C 180,E1 -18176.769,E2 -18176.769} C_VEL
LIN {X 0,Y 278.403,Z 371.019,A -85,B 0,C 180,E1 -18178.191,E2 -18178.191} C_VEL
LIN {X 0,Y 276.268,Z 379.169,A -85,B 0,C 180,E1 -18179.635,E2 -18179.635} C_VEL
LIN {X 0,Y 273.763,Z 387.433,A -85,B 0,C 180,E1 -18181.47,E2 -18181.47} C_VEL
LIN {X 0,Y 271.566,Z 394.099,A -85,B 0,C 180,E1 -18183.337,E2 -18183.337} C_VEL
LIN {X 0,Y 269.511,Z 399.463,A -85,B 0,C 180,E1 -18185.236,E2 -18185.236} C_VEL
LIN {X 0,Y 267.435,Z 404.319,A -85,B 0,C 180,E1 -18187.55,E2 -18187.55} C_VEL
LIN {X 0,Y 266.245,Z 406.772,A -85,B 0,C 180,E1 -18189.112,E2 -18189.112} C_VEL
LIN {X 0,Y 264.984,Z 408.984,A -85,B 0,C 180,E1 -18191.087,E2 -18191.087} C_VEL
LIN {X 0,Y 264.31,Z 409.883,A -85,B 0,C 180,E1 -18192.281,E2 -18192.281} C_VEL
LIN {X 0,Y 263.559,Z 410.614,A -85,B 0,C 180,E1 -18193.885,E2 -18193.885} C_VEL
LIN {X 0,Y 262.876,Z 410.724,A -85,B 0,C 180,E1 -18195.747,E2 -18195.747} C_VEL
LIN {X 0,Y 262.451,Z 410.34,A -85,B 0,C 180,E1 -18197.13,E2 -18197.13} C_VEL
LIN {X 0,Y 262.12,Z 409.337,A -85,B 0,C 180,E1 -18198.768,E2 -18198.768} C_VEL
LIN {X 0,Y 261.87,Z 406.729,A -85,B 0,C 180,E1 -18201.241,E2 -18201.241} C_VEL
LIN {X 0,Y 261.989,Z 402.672,A -85,B 0,C 180,E1 -18203.726,E2 -18203.726} C_VEL
LIN {X 0,Y 262.357,Z 396.925,A -85,B 0,C 180,E1 -18206.231,E2 -18206.231} C_VEL
LIN {X 0,Y 262.799,Z 390.67,A -85,B 0,C 180,E1 -18208.326,E2 -18208.326} C_VEL
LIN {X 0,Y 263.363,Z 382.532,A -85,B 0,C 180,E1 -18210.465,E2 -18210.465} C_VEL
LIN {X 0,Y 264.181,Z 373.384,A -85,B 0,C 180,E1 -18212.369,E2 -18212.369} C_VEL
LIN {X 0,Y 264.959,Z 363.425,A -85,B 0,C 180,E1 -18214.024,E2 -18214.024} C_VEL
LIN {X 0,Y 265.843,Z 351.529,A -85,B 0,C 180,E1 -18215.563,E2 -18215.563} C_VEL
LIN {X 0,Y 266.564,Z 339.486,A -85,B 0,C 180,E1 -18216.737,E2 -18216.737} C_VEL
LIN {X 0,Y 267.137,Z 326.801,A -85,B 0,C 180,E1 -18217.628,E2 -18217.628} C_VEL
LIN {X 0,Y 267.462,Z 313.617,A -85,B 0,C 180,E1 -18218.234,E2 -18218.234} C_VEL
LIN {X 0,Y 269.143,Z 259.027,A -85,B 0,C 180,E1 -18220.259,E2 -18220.259} C_VEL
LIN {X 0,Y 265.992,Z 234.284,A -85,B 0,C 180,E1 -18221.391,E2 -18221.391} C_VEL
LIN {X 0,Y 266.307,Z 229.316,A -85,B 0,C 180,E1 -18222.748,E2 -18222.748} C_VEL
LIN {X 0,Y 265.918,Z 225.653,A -85,B 0,C 180,E1 -18223.87,E2 -18223.87} C_VEL
LIN {X 0,Y 263.872,Z 215.16,A -85,B 0,C 180,E1 -18227.22,E2 -18227.22} C_VEL
LIN {X 0,Y 263.18,Z 211.839,A -85,B 0,C 180,E1 -18228.392,E2 -18228.392} C_VEL
LIN {X 0,Y 263.182,Z 211.702,A -85,B 0,C 180,E1 -18233.236,E2 -18233.236} C_VEL
LIN {X 0,Y 263.167,Z 211.705,A -85,B 0,C 180,E1 -18235.887,E2 -18235.887} C_VEL
LIN {X 0,Y 263.15,Z 211.708,A -85,B 0,C 180,E1 -18239.506,E2 -18239.506} C_VEL
LIN {X 0,Y 263.192,Z 211.7,A -85,B 0,C 180,E1 -18243.002,E2 -18243.002} C_VEL
LIN {X 0,Y 263.183,Z 211.699,A -85,B 0,C 180,E1 -18246.386,E2 -18246.386} C_VEL
LIN {X 0,Y 263.262,Z 211.692,A -85,B 0,C 180,E1 -18249.692,E2 -18249.692} C_VEL
LIN {X 0,Y 263.349,Z 211.678,A -85,B 0,C 180,E1 -18254.521,E2 -18254.521} C_VEL
LIN {X 0,Y 263.372,Z 211.68,A -85,B 0,C 180,E1 -18259.233,E2 -18259.233} C_VEL
LIN {X 0,Y 263.571,Z 211.65,A -85,B 0,C 180,E1 -18262.337,E2 -18262.337} C_VEL
LIN {X 0,Y 263.749,Z 211.629,A -85,B 0,C 180,E1 -18268.472,E2 -18268.472} C_VEL
LIN {X 0,Y 263.749,Z 211.63,A -85,B 0,C 180,E1 -18271.526,E2 -18271.526} C_VEL
LIN {X 0,Y 263.566,Z 211.65,A -85,B 0,C 180,E1 -18277.661,E2 -18277.661} C_VEL
LIN {X 0,Y 263.37,Z 211.679,A -85,B 0,C 180,E1 -18280.765,E2 -18280.765} C_VEL
LIN {X 0,Y 263.347,Z 211.678,A -85,B 0,C 180,E1 -18285.477,E2 -18285.477} C_VEL
LIN {X 0,Y 263.259,Z 211.691,A -85,B 0,C 180,E1 -18290.306,E2 -18290.306} C_VEL
LIN {X 0,Y 263.204,Z 211.696,A -85,B 0,C 180,E1 -18295.29,E2 -18295.29} C_VEL
LIN {X 0,Y 263.175,Z 211.704,A -85,B 0,C 180,E1 -18298.729,E2 -18298.729} C_VEL
LIN {X 0,Y 263.128,Z 211.708,A -85,B 0,C 180,E1 -18302.287,E2 -18302.287} C_VEL
LIN {X 0,Y 263.184,Z 211.7,A -85,B 0,C 180,E1 -18305.977,E2 -18305.977} C_VEL
LIN {X 0,Y 263.153,Z 211.703,A -85,B 0,C 180,E1 -18309.862,E2 -18309.862} C_VEL
LIN {X 0,Y 263.139,Z 211.706,A -85,B 0,C 180,E1 -18313.979,E2 -18313.979} C_VEL
LIN {X 0,Y 263.15,Z 211.706,A -85,B 0,C 180,E1 -18318.398,E2 -18318.398} C_VEL
LIN {X 0,Y 263.199,Z 211.697,A -85,B 0,C 180,E1 -18323.23,E2 -18323.23} C_VEL
LIN {X 0,Y 263.176,Z 211.702,A -85,B 0,C 180,E1 -18325.89,E2 -18325.89} C_VEL
LIN {X 0,Y 263.141,Z 211.704,A -85,B 0,C 180,E1 -18329.507,E2 -18329.507} C_VEL
LIN {X 0,Y 263.185,Z 211.699,A -85,B 0,C 180,E1 -18333.003,E2 -18333.003} C_VEL
LIN {X 0,Y 263.176,Z 211.7,A -85,B 0,C 180,E1 -18336.387,E2 -18336.387} C_VEL
LIN {X 0,Y 263.256,Z 211.692,A -85,B 0,C 180,E1 -18339.694,E2 -18339.694} C_VEL
LIN {X 0,Y 263.343,Z 211.678,A -85,B 0,C 180,E1 -18344.522,E2 -18344.522} C_VEL
LIN {X 0,Y 263.348,Z 211.68,A -85,B 0,C 180,E1 -18349.234,E2 -18349.234} C_VEL
LIN {X 0,Y 263.551,Z 211.653,A -85,B 0,C 180,E1 -18352.339,E2 -18352.339} C_VEL
LIN {X 0,Y 263.744,Z 211.63,A -85,B 0,C 180,E1 -18358.474,E2 -18358.474} C_VEL
LIN {X 0,Y 263.744,Z 211.632,A -85,B 0,C 180,E1 -18361.528,E2 -18361.528} C_VEL
LIN {X 0,Y 263.566,Z 211.655,A -85,B 0,C 180,E1 -18367.663,E2 -18367.663} C_VEL
LIN {X 0,Y 263.424,Z 211.667,A -85,B 0,C 180,E1 -18370.072,E2 -18370.072} C_VEL
LIN {X 0,Y 262.671,Z 211.764,A -85,B 0,C 180,E1 -18371.347,E2 -18371.347} C_VEL
LIN {X 0,Y 259.8,Z 212.125,A -85,B 0,C 180,E1 -18373.426,E2 -18373.426} C_VEL
LIN {X 0,Y 257.394,Z 212.423,A -85,B 0,C 180,E1 -18375.116,E2 -18375.116} C_VEL
LIN {X 0,Y 256.334,Z 212.552,A -85,B 0,C 180,E1 -18376.426,E2 -18376.426} C_VEL
LIN {X 0,Y 256.229,Z 212.564,A -85,B 0,C 180,E1 -18376.87,E2 -18376.87} C_VEL
LIN {X 0,Y 256.152,Z 212.577,A -85,B 0,C 180,E1 -18381.121,E2 -18381.121} C_VEL
LIN {X 0,Y 256.183,Z 212.575,A -85,B 0,C 180,E1 -18385.14,E2 -18385.14} C_VEL
LIN {X 0,Y 256.099,Z 212.584,A -85,B 0,C 180,E1 -18389.602,E2 -18389.602} C_VEL
LIN {X 0,Y 256.064,Z 212.59,A -85,B 0,C 180,E1 -18393.294,E2 -18393.294} C_VEL
LIN {X 0,Y 256.111,Z 212.584,A -85,B 0,C 180,E1 -18397.272,E2 -18397.272} C_VEL
LIN {X 0,Y 256.052,Z 212.592,A -85,B 0,C 180,E1 -18401.205,E2 -18401.205} C_VEL
LIN {X 0,Y 256.038,Z 212.591,A -85,B 0,C 180,E1 -18405.536,E2 -18405.536} C_VEL
LIN {X 0,Y 256.053,Z 212.592,A -85,B 0,C 180,E1 -18408.798,E2 -18408.798} C_VEL
LIN {X 0,Y 256.162,Z 212.766,A -85,B 0,C 180,E1 -18413.059,E2 -18413.059} C_VEL
LIN {X 0,Y 259.365,Z 227.027,A -85,B 0,C 180,E1 -18417.186,E2 -18417.186} C_VEL
LIN {X 0,Y 262.164,Z 239.893,A -85,B 0,C 180,E1 -18420.711,E2 -18420.711} C_VEL
LIN {X 0,Y 262.056,Z 243.238,A -85,B 0,C 180,E1 -18421.557,E2 -18421.557} C_VEL
LIN {X 0,Y 259.91,Z 256.954,A -85,B 0,C 180,E1 -18424.897,E2 -18424.897} C_VEL
LIN {X 0,Y 261.173,Z 279.693,A -85,B 0,C 180,E1 -18425.826,E2 -18425.826} C_VEL
LIN {X 0,Y 262.734,Z 299.203,A -85,B 0,C 180,E1 -18426.602,E2 -18426.602} C_VEL
LIN {X 0,Y 261.003,Z 360.341,A -85,B 0,C 180,E1 -18428.737,E2 -18428.737} C_VEL
LIN {X 0,Y 260.31,Z 372.793,A -85,B 0,C 180,E1 -18429.454,E2 -18429.454} C_VEL
LIN {X 0,Y 259.421,Z 384.508,A -85,B 0,C 180,E1 -18430.414,E2 -18430.414} C_VEL
LIN {X 0,Y 258.345,Z 396.773,A -85,B 0,C 180,E1 -18431.771,E2 -18431.771} C_VEL
LIN {X 0,Y 257.34,Z 407.294,A -85,B 0,C 180,E1 -18433.261,E2 -18433.261} C_VEL
LIN {X 0,Y 256.36,Z 416.578,A -85,B 0,C 180,E1 -18434.905,E2 -18434.905} C_VEL
LIN {X 0,Y 255.605,Z 425.676,A -85,B 0,C 180,E1 -18436.89,E2 -18436.89} C_VEL
LIN {X 0,Y 255.108,Z 433.108,A -85,B 0,C 180,E1 -18438.882,E2 -18438.882} C_VEL
LIN {X 0,Y 254.856,Z 440.256,A -85,B 0,C 180,E1 -18441.277,E2 -18441.277} C_VEL
LIN {X 0,Y 254.855,Z 445.829,A -85,B 0,C 180,E1 -18443.668,E2 -18443.668} C_VEL
LIN {X 0,Y 254.966,Z 450.039,A -85,B 0,C 180,E1 -18446.05,E2 -18446.05} C_VEL
LIN {X 0,Y 255.193,Z 453.026,A -85,B 0,C 180,E1 -18448.423,E2 -18448.423} C_VEL
LIN {X 0,Y 255.186,Z 454.362,A -85,B 0,C 180,E1 -18450.001,E2 -18450.001} C_VEL
LIN {X 0,Y 255.105,Z 455.194,A -85,B 0,C 180,E1 -18451.58,E2 -18451.58} C_VEL
LIN {X 0,Y 254.728,Z 455.56,A -85,B 0,C 180,E1 -18453.164,E2 -18453.164} C_VEL
LIN {X 0,Y 254.42,Z 455.132,A -85,B 0,C 180,E1 -18456.034,E2 -18456.034} C_VEL
LIN {X 0,Y 254.348,Z 454.064,A -85,B 0,C 180,E1 -18457.942,E2 -18457.942} C_VEL
LIN {X 0,Y 254.495,Z 452.74,A -85,B 0,C 180,E1 -18459.538,E2 -18459.538} C_VEL
LIN {X 0,Y 254.999,Z 449.907,A -85,B 0,C 180,E1 -18461.93,E2 -18461.93} C_VEL
LIN {X 0,Y 256.163,Z 446.085,A -85,B 0,C 180,E1 -18464.296,E2 -18464.296} C_VEL
LIN {X 0,Y 257.7,Z 441.145,A -85,B 0,C 180,E1 -18466.641,E2 -18466.641} C_VEL
LIN {X 0,Y 260.096,Z 433.768,A -85,B 0,C 180,E1 -18469.331,E2 -18469.331} C_VEL
LIN {X 0,Y 262.736,Z 425.844,A -85,B 0,C 180,E1 -18471.581,E2 -18471.581} C_VEL
LIN {X 0,Y 266.031,Z 416.027,A -85,B 0,C 180,E1 -18473.759,E2 -18473.759} C_VEL
LIN {X 0,Y 268.717,Z 407.052,A -85,B 0,C 180,E1 -18475.359,E2 -18475.359} C_VEL
LIN {X 0,Y 271.808,Z 395.991,A -85,B 0,C 180,E1 -18476.904,E2 -18476.904} C_VEL
LIN {X 0,Y 274.448,Z 385.294,A -85,B 0,C 180,E1 -18478.07,E2 -18478.07} C_VEL
LIN {X 0,Y 277.068,Z 372.551,A -85,B 0,C 180,E1 -18479.125,E2 -18479.125} C_VEL
LIN {X 0,Y 279.16,Z 359.251,A -85,B 0,C 180,E1 -18479.921,E2 -18479.921} C_VEL
LIN {X 0,Y 280.598,Z 343.796,A -85,B 0,C 180,E1 -18480.539,E2 -18480.539} C_VEL
LIN {X 0,Y 283.642,Z 304.927,A -85,B 0,C 180,E1 -18481.929,E2 -18481.929} C_VEL
LIN {X 0,Y 282.957,Z 290.661,A -85,B 0,C 180,E1 -18482.853,E2 -18482.853} C_VEL
LIN {X 0,Y 281.265,Z 274.397,A -85,B 0,C 180,E1 -18484.196,E2 -18484.196} C_VEL
LIN {X 0,Y 280.528,Z 269.759,A -85,B 0,C 180,E1 -18484.651,E2 -18484.651} C_VEL
LIN {X 0,Y 276.494,Z 261.081,A -85,B 0,C 180,E1 -18486.296,E2 -18486.296} C_VEL
LIN {X 0,Y 273.716,Z 255.821,A -85,B 0,C 180,E1 -18487.486,E2 -18487.486} C_VEL
LIN {X 0,Y 271.162,Z 250.969,A -85,B 0,C 180,E1 -18488.769,E2 -18488.769} C_VEL
LIN {X 0,Y 269.855,Z 246.538,A -85,B 0,C 180,E1 -18490.951,E2 -18490.951} C_VEL
LIN {X 0,Y 268.445,Z 241.912,A -85,B 0,C 180,E1 -18493.635,E2 -18493.635} C_VEL
LIN {X 0,Y 266.96,Z 237.564,A -85,B 0,C 180,E1 -18496.805,E2 -18496.805} C_VEL
LIN {X 0,Y 265.709,Z 234.215,A -85,B 0,C 180,E1 -18500.091,E2 -18500.091} C_VEL
LIN {X 0,Y 264.972,Z 232.333,A -85,B 0,C 180,E1 -18502.723,E2 -18502.723} C_VEL
LIN {X 0,Y 264.39,Z 230.997,A -85,B 0,C 180,E1 -18506.066,E2 -18506.066} C_VEL
LIN {X 0,Y 264.254,Z 230.755,A -85,B 0,C 180,E1 -18509.647,E2 -18509.647} C_VEL
LIN {X 0,Y 264.752,Z 231.622,A -85,B 0,C 180,E1 -18513.174,E2 -18513.174} C_VEL
LIN {X 0,Y 265.488,Z 233.828,A -85,B 0,C 180,E1 -18516.604,E2 -18516.604} C_VEL
LIN {X 0,Y 266.667,Z 237.001,A -85,B 0,C 180,E1 -18519.963,E2 -18519.963} C_VEL
LIN {X 0,Y 268.033,Z 240.999,A -85,B 0,C 180,E1 -18523.021,E2 -18523.021} C_VEL
LIN {X 0,Y 272.215,Z 247.179,A -85,B 0,C 180,E1 -18525.149,E2 -18525.149} C_VEL
LIN {X 0,Y 275.603,Z 252.413,A -85,B 0,C 180,E1 -18526.654,E2 -18526.654} C_VEL
LIN {X 0,Y 279.965,Z 259.868,A -85,B 0,C 180,E1 -18528.441,E2 -18528.441} C_VEL
LIN {X 0,Y 284.381,Z 269.114,A -85,B 0,C 180,E1 -18530.146,E2 -18530.146} C_VEL
LIN {X 0,Y 285.37,Z 275.358,A -85,B 0,C 180,E1 -18530.777,E2 -18530.777} C_VEL
LIN {X 0,Y 280.482,Z 326.976,A -85,B 0,C 180,E1 -18532.893,E2 -18532.893} C_VEL
LIN {X 0,Y 279.06,Z 339.62,A -85,B 0,C 180,E1 -18533.673,E2 -18533.673} C_VEL
LIN {X 0,Y 277.232,Z 351.264,A -85,B 0,C 180,E1 -18534.677,E2 -18534.677} C_VEL
LIN {X 0,Y 274.972,Z 362.539,A -85,B 0,C 180,E1 -18535.965,E2 -18535.965} C_VEL
LIN {X 0,Y 272.248,Z 373.541,A -85,B 0,C 180,E1 -18537.595,E2 -18537.595} C_VEL
LIN {X 0,Y 269.746,Z 382.243,A -85,B 0,C 180,E1 -18539.253,E2 -18539.253} C_VEL
LIN {X 0,Y 267.121,Z 390.191,A -85,B 0,C 180,E1 -18541.16,E2 -18541.16} C_VEL
LIN {X 0,Y 264.374,Z 397.414,A -85,B 0,C 180,E1 -18543.428,E2 -18543.428} C_VEL
LIN {X 0,Y 262.323,Z 402.205,A -85,B 0,C 180,E1 -18545.38,E2 -18545.38} C_VEL
LIN {X 0,Y 260.219,Z 406.518,A -85,B 0,C 180,E1 -18547.76,E2 -18547.76} C_VEL
LIN {X 0,Y 259.006,Z 408.645,A -85,B 0,C 180,E1 -18549.369,E2 -18549.369} C_VEL
LIN {X 0,Y 257.885,Z 410.271,A -85,B 0,C 180,E1 -18551.158,E2 -18551.158} C_VEL
LIN {X 0,Y 257.053,Z 411.104,A -85,B 0,C 180,E1 -18552.633,E2 -18552.633} C_VEL
LIN {X 0,Y 256.307,Z 411.502,A -85,B 0,C 180,E1 -18554.286,E2 -18554.286} C_VEL
LIN {X 0,Y 255.731,Z 411.332,A -85,B 0,C 180,E1 -18555.95,E2 -18555.95} C_VEL
LIN {X 0,Y 255.264,Z 410.618,A -85,B 0,C 180,E1 -18557.628,E2 -18557.628} C_VEL
LIN {X 0,Y 254.854,Z 408.189,A -85,B 0,C 180,E1 -18560.346,E2 -18560.346} C_VEL
LIN {X 0,Y 254.803,Z 404.818,A -85,B 0,C 180,E1 -18562.714,E2 -18562.714} C_VEL
LIN {X 0,Y 255.092,Z 399.636,A -85,B 0,C 180,E1 -18565.278,E2 -18565.278} C_VEL
LIN {X 0,Y 255.483,Z 393.928,A -85,B 0,C 180,E1 -18567.436,E2 -18567.436} C_VEL
LIN {X 0,Y 256.014,Z 386.582,A -85,B 0,C 180,E1 -18569.611,E2 -18569.611} C_VEL
LIN {X 0,Y 256.73,Z 377.839,A -85,B 0,C 180,E1 -18571.664,E2 -18571.664} C_VEL
LIN {X 0,Y 257.574,Z 367.759,A -85,B 0,C 180,E1 -18573.54,E2 -18573.54} C_VEL
LIN {X 0,Y 258.424,Z 357.031,A -85,B 0,C 180,E1 -18575.107,E2 -18575.107} C_VEL
LIN {X 0,Y 259.224,Z 345.534,A -85,B 0,C 180,E1 -18576.41,E2 -18576.41} C_VEL
LIN {X 0,Y 259.805,Z 334.431,A -85,B 0,C 180,E1 -18577.369,E2 -18577.369} C_VEL
LIN {X 0,Y 260.287,Z 321.084,A -85,B 0,C 180,E1 -18578.174,E2 -18578.174} C_VEL
LIN {X 0,Y 262.176,Z 259.248,A -85,B 0,C 180,E1 -18580.569,E2 -18580.569} C_VEL
LIN {X 0,Y 259.047,Z 234.66,A -85,B 0,C 180,E1 -18581.727,E2 -18581.727} C_VEL
LIN {X 0,Y 259.256,Z 231.137,A -85,B 0,C 180,E1 -18582.664,E2 -18582.664} C_VEL
LIN {X 0,Y 258.931,Z 226.831,A -85,B 0,C 180,E1 -18584.005,E2 -18584.005} C_VEL
LIN {X 0,Y 256.726,Z 215.675,A -85,B 0,C 180,E1 -18587.657,E2 -18587.657} C_VEL
LIN {X 0,Y 256.172,Z 212.921,A -85,B 0,C 180,E1 -18588.61,E2 -18588.61} C_VEL
LIN {X 0,Y 256.114,Z 212.584,A -85,B 0,C 180,E1 -18589.198,E2 -18589.198} C_VEL
LIN {X 0,Y 256.13,Z 212.58,A -85,B 0,C 180,E1 -18592.866,E2 -18592.866} C_VEL
LIN {X 0,Y 256.076,Z 212.585,A -85,B 0,C 180,E1 -18596.707,E2 -18596.707} C_VEL
LIN {X 0,Y 256.138,Z 212.581,A -85,B 0,C 180,E1 -18601.404,E2 -18601.404} C_VEL
LIN {X 0,Y 256.166,Z 212.576,A -85,B 0,C 180,E1 -18605.698,E2 -18605.698} C_VEL
LIN {X 0,Y 256.165,Z 212.576,A -85,B 0,C 180,E1 -18609.104,E2 -18609.104} C_VEL
LIN {X 0,Y 256.298,Z 212.556,A -85,B 0,C 180,E1 -18614.084,E2 -18614.084} C_VEL
LIN {X 0,Y 256.308,Z 212.558,A -85,B 0,C 180,E1 -18618.933,E2 -18618.933} C_VEL
LIN {X 0,Y 256.538,Z 212.526,A -85,B 0,C 180,E1 -18622.126,E2 -18622.126} C_VEL
LIN {X 0,Y 256.712,Z 212.505,A -85,B 0,C 180,E1 -18628.43,E2 -18628.43} C_VEL
LIN {X 0,Y 256.712,Z 212.506,A -85,B 0,C 180,E1 -18631.568,E2 -18631.568} C_VEL
LIN {X 0,Y 256.534,Z 212.525,A -85,B 0,C 180,E1 -18637.872,E2 -18637.872} C_VEL
LIN {X 0,Y 256.306,Z 212.559,A -85,B 0,C 180,E1 -18641.065,E2 -18641.065} C_VEL
LIN {X 0,Y 256.296,Z 212.556,A -85,B 0,C 180,E1 -18645.914,E2 -18645.914} C_VEL
LIN {X 0,Y 256.162,Z 212.577,A -85,B 0,C 180,E1 -18650.894,E2 -18650.894} C_VEL
LIN {X 0,Y 256.184,Z 212.571,A -85,B 0,C 180,E1 -18655.138,E2 -18655.138} C_VEL
LIN {X 0,Y 256.109,Z 212.581,A -85,B 0,C 180,E1 -18659.599,E2 -18659.599} C_VEL
LIN {X 0,Y 256.079,Z 212.583,A -85,B 0,C 180,E1 -18663.289,E2 -18663.289} C_VEL
LIN {X 0,Y 256.135,Z 212.578,A -85,B 0,C 180,E1 -18667.278,E2 -18667.278} C_VEL
LIN {X 0,Y 256.097,Z 212.58,A -85,B 0,C 180,E1 -18671.193,E2 -18671.193} C_VEL
LIN {X 0,Y 256.069,Z 212.586,A -85,B 0,C 180,E1 -18675.525,E2 -18675.525} C_VEL
LIN {X 0,Y 256.08,Z 212.584,A -85,B 0,C 180,E1 -18678.803,E2 -18678.803} C_VEL
LIN {X 0,Y 256.148,Z 212.576,A -85,B 0,C 180,E1 -18682.871,E2 -18682.871} C_VEL
LIN {X 0,Y 256.078,Z 212.584,A -85,B 0,C 180,E1 -18686.71,E2 -18686.71} C_VEL
LIN {X 0,Y 256.128,Z 212.578,A -85,B 0,C 180,E1 -18691.406,E2 -18691.406} C_VEL
LIN {X 0,Y 256.16,Z 212.575,A -85,B 0,C 180,E1 -18695.699,E2 -18695.699} C_VEL
LIN {X 0,Y 256.159,Z 212.574,A -85,B 0,C 180,E1 -18699.105,E2 -18699.105} C_VEL
LIN {X 0,Y 256.293,Z 212.559,A -85,B 0,C 180,E1 -18704.085,E2 -18704.085} C_VEL
LIN {X 0,Y 256.29,Z 212.558,A -85,B 0,C 180,E1 -18708.934,E2 -18708.934} C_VEL
LIN {X 0,Y 256.508,Z 212.532,A -85,B 0,C 180,E1 -18712.127,E2 -18712.127} C_VEL
LIN {X 0,Y 256.491,Z 212.533,A -85,B 0,C 180,E1 -18716.859,E2 -18716.859} C_VEL
LIN {X 0,Y 256.759,Z 212.501,A -85,B 0,C 180,E1 -18720.001,E2 -18720.001} C_VEL
LIN {X 0,Y 256.491,Z 212.532,A -85,B 0,C 180,E1 -18723.142,E2 -18723.142} C_VEL
LIN {X 0,Y 256.533,Z 212.529,A -85,B 0,C 180,E1 -18727.874,E2 -18727.874} C_VEL
LIN {X 0,Y 256.304,Z 212.555,A -85,B 0,C 180,E1 -18731.067,E2 -18731.067} C_VEL
LIN {X 0,Y 256.294,Z 212.558,A -85,B 0,C 180,E1 -18735.916,E2 -18735.916} C_VEL
LIN {X 0,Y 256.229,Z 212.564,A -85,B 0,C 180,E1 -18736.87,E2 -18736.87} C_VEL
LIN {X 0,Y 255.5,Z 212.657,A -85,B 0,C 180,E1 -18738.182,E2 -18738.182} C_VEL
LIN {X 0,Y 252.591,Z 213.024,A -85,B 0,C 180,E1 -18740.32,E2 -18740.32} C_VEL
LIN {X 0,Y 250.165,Z 213.326,A -85,B 0,C 180,E1 -18742.06,E2 -18742.06} C_VEL
LIN {X 0,Y 249.146,Z 213.452,A -85,B 0,C 180,E1 -18743.41,E2 -18743.41} C_VEL
LIN {X 0,Y 249.073,Z 213.457,A -85,B 0,C 180,E1 -18743.868,E2 -18743.868} C_VEL
LIN {X 0,Y 249.067,Z 213.458,A -85,B 0,C 180,E1 -18746.839,E2 -18746.839} C_VEL
LIN {X 0,Y 249.043,Z 213.461,A -85,B 0,C 180,E1 -18750.529,E2 -18750.529} C_VEL
LIN {X 0,Y 249.041,Z 213.466,A -85,B 0,C 180,E1 -18755.079,E2 -18755.079} C_VEL
LIN {X 0,Y 249.022,Z 213.464,A -85,B 0,C 180,E1 -18758.382,E2 -18758.382} C_VEL
LIN {X 0,Y 248.998,Z 213.47,A -85,B 0,C 180,E1 -18762.792,E2 -18762.792} C_VEL
LIN {X 0,Y 249.007,Z 213.468,A -85,B 0,C 180,E1 -18767.363,E2 -18767.363} C_VEL
LIN {X 0,Y 249.049,Z 213.463,A -85,B 0,C 180,E1 -18772.2,E2 -18772.2} C_VEL
LIN {X 0,Y 249.167,Z 213.889,A -85,B 0,C 180,E1 -18772.738,E2 -18772.738} C_VEL
LIN {X 0,Y 252.58,Z 229.109,A -85,B 0,C 180,E1 -18777.246,E2 -18777.246} C_VEL
LIN {X 0,Y 255.208,Z 241.568,A -85,B 0,C 180,E1 -18780.74,E2 -18780.74} C_VEL
LIN {X 0,Y 254.291,Z 248.351,A -85,B 0,C 180,E1 -18782.462,E2 -18782.462} C_VEL
LIN {X 0,Y 252.957,Z 256.75,A -85,B 0,C 180,E1 -18784.548,E2 -18784.548} C_VEL
LIN {X 0,Y 254.427,Z 283.355,A -85,B 0,C 180,E1 -18785.656,E2 -18785.656} C_VEL
LIN {X 0,Y 255.746,Z 299.749,A -85,B 0,C 180,E1 -18786.33,E2 -18786.33} C_VEL
LIN {X 0,Y 254.016,Z 359.803,A -85,B 0,C 180,E1 -18788.496,E2 -18788.496} C_VEL
LIN {X 0,Y 253.252,Z 372.923,A -85,B 0,C 180,E1 -18789.28,E2 -18789.28} C_VEL
LIN {X 0,Y 252.35,Z 384.412,A -85,B 0,C 180,E1 -18790.266,E2 -18790.266} C_VEL
LIN {X 0,Y 251.271,Z 396.584,A -85,B 0,C 180,E1 -18791.661,E2 -18791.661} C_VEL
LIN {X 0,Y 250.305,Z 406.55,A -85,B 0,C 180,E1 -18793.117,E2 -18793.117} C_VEL
LIN {X 0,Y 249.277,Z 416.24,A -85,B 0,C 180,E1 -18794.884,E2 -18794.884} C_VEL
LIN {X 0,Y 248.515,Z 425.291,A -85,B 0,C 180,E1 -18796.926,E2 -18796.926} C_VEL
LIN {X 0,Y 248.026,Z 432.682,A -85,B 0,C 180,E1 -18798.975,E2 -18798.975} C_VEL
LIN {X 0,Y 247.818,Z 439.769,A -85,B 0,C 180,E1 -18801.439,E2 -18801.439} C_VEL
LIN {X 0,Y 247.798,Z 444.469,A -85,B 0,C 180,E1 -18803.487,E2 -18803.487} C_VEL
LIN {X 0,Y 247.943,Z 448.832,A -85,B 0,C 180,E1 -18805.938,E2 -18805.938} C_VEL
LIN {X 0,Y 248.15,Z 451.952,A -85,B 0,C 180,E1 -18808.378,E2 -18808.378} C_VEL
LIN {X 0,Y 248.148,Z 453.392,A -85,B 0,C 180,E1 -18810.001,E2 -18810.001} C_VEL
LIN {X 0,Y 248.05,Z 454.319,A -85,B 0,C 180,E1 -18811.625,E2 -18811.625} C_VEL
LIN {X 0,Y 247.675,Z 454.754,A -85,B 0,C 180,E1 -18813.254,E2 -18813.254} C_VEL
LIN {X 0,Y 247.344,Z 454.536,A -85,B 0,C 180,E1 -18816.013,E2 -18816.013} C_VEL
LIN {X 0,Y 247.294,Z 453.519,A -85,B 0,C 180,E1 -18818.17,E2 -18818.17} C_VEL
LIN {X 0,Y 247.754,Z 450.618,A -85,B 0,C 180,E1 -18821.454,E2 -18821.454} C_VEL
LIN {X 0,Y 248.811,Z 447.293,A -85,B 0,C 180,E1 -18823.893,E2 -18823.893} C_VEL
